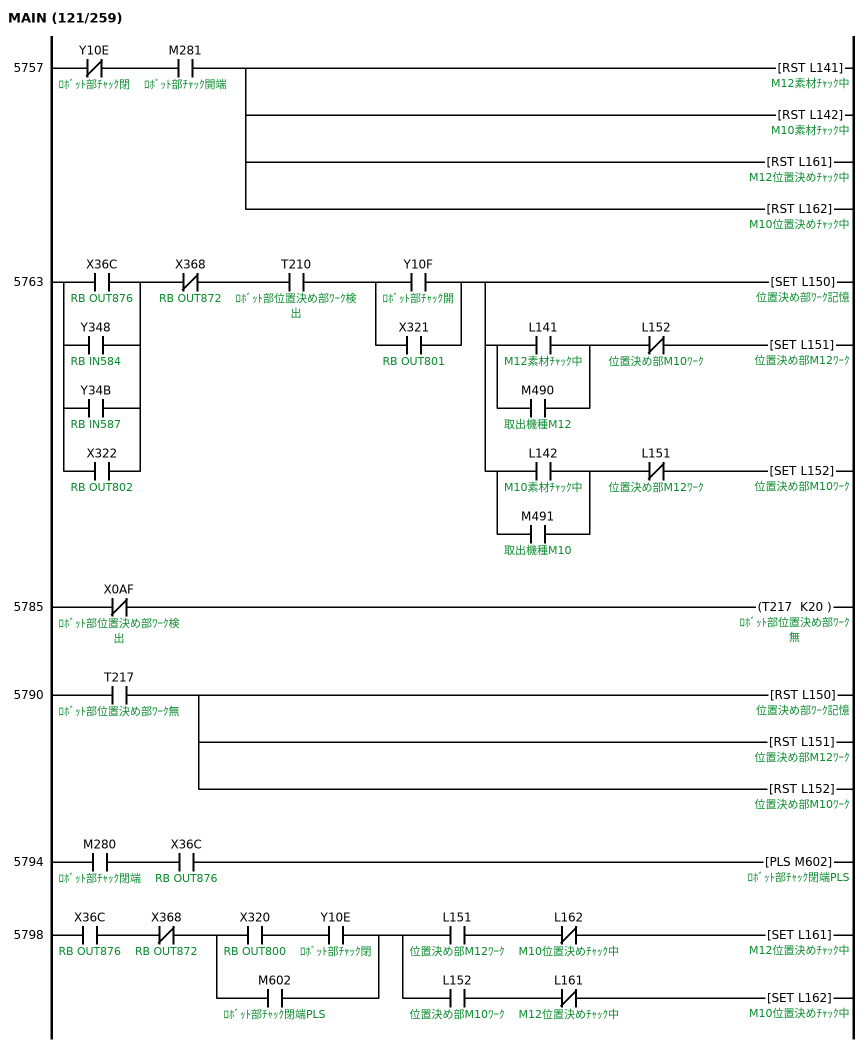
[picture p120: ladder of MAIN, rungs at steps 5757 to 5798]
5757  LDI     Y10E  ; ﾛﾎﾞｯﾄ部ﾁｬｯｸ閉
      AND     M281  ; ﾛﾎﾞｯﾄ部ﾁｬｯｸ開端
      RST     L141  ; M12素材ﾁｬｯｸ中
      RST     L142  ; M10素材ﾁｬｯｸ中
      RST     L161  ; M12位置決めﾁｬｯｸ中
      RST     L162  ; M10位置決めﾁｬｯｸ中
5763  LD      X36C  ; RB OUT876
      OR      Y348  ; RB IN584
      OR      Y34B  ; RB IN587
      OR      X322  ; RB OUT802
      ANI     X368  ; RB OUT872
      AND     T210  ; ﾛﾎﾞｯﾄ部位置決め部ﾜｰｸ検出
      LD      Y10F  ; ﾛﾎﾞｯﾄ部ﾁｬｯｸ開
      OR      X321  ; RB OUT801
      ANB
      SET     L150  ; 位置決め部ﾜｰｸ記憶
      MPS
      LD      L141  ; M12素材ﾁｬｯｸ中
      OR      M490  ; 取出機種M12
      ANB
      ANI     L152  ; 位置決め部M10ﾜｰｸ
      SET     L151  ; 位置決め部M12ﾜｰｸ
      MPP
      LD      L142  ; M10素材ﾁｬｯｸ中
      OR      M491  ; 取出機種M10
      ANB
      ANI     L151  ; 位置決め部M12ﾜｰｸ
      SET     L152  ; 位置決め部M10ﾜｰｸ
5785  LDI     X0AF  ; ﾛﾎﾞｯﾄ部位置決め部ﾜｰｸ検出
      OUT     T217 K20  ; ﾛﾎﾞｯﾄ部位置決め部ﾜｰｸ無
5790  LD      T217  ; ﾛﾎﾞｯﾄ部位置決め部ﾜｰｸ無
      RST     L150  ; 位置決め部ﾜｰｸ記憶
      RST     L151  ; 位置決め部M12ﾜｰｸ
      RST     L152  ; 位置決め部M10ﾜｰｸ
5794  LD      M280  ; ﾛﾎﾞｯﾄ部ﾁｬｯｸ閉端
      AND     X36C  ; RB OUT876
      PLS     M602  ; ﾛﾎﾞｯﾄ部ﾁｬｯｸ閉端PLS
5798  LD      X36C  ; RB OUT876
      ANI     X368  ; RB OUT872
      LD      X320  ; RB OUT800
      AND     Y10E  ; ﾛﾎﾞｯﾄ部ﾁｬｯｸ閉
      OR      M602  ; ﾛﾎﾞｯﾄ部ﾁｬｯｸ閉端PLS
      ANB
      MPS
      AND     L151  ; 位置決め部M12ﾜｰｸ
      ANI     L162  ; M10位置決めﾁｬｯｸ中
      SET     L161  ; M12位置決めﾁｬｯｸ中
      MPP
      AND     L152  ; 位置決め部M10ﾜｰｸ
      ANI     L161  ; M12位置決めﾁｬｯｸ中
      SET     L162  ; M10位置決めﾁｬｯｸ中
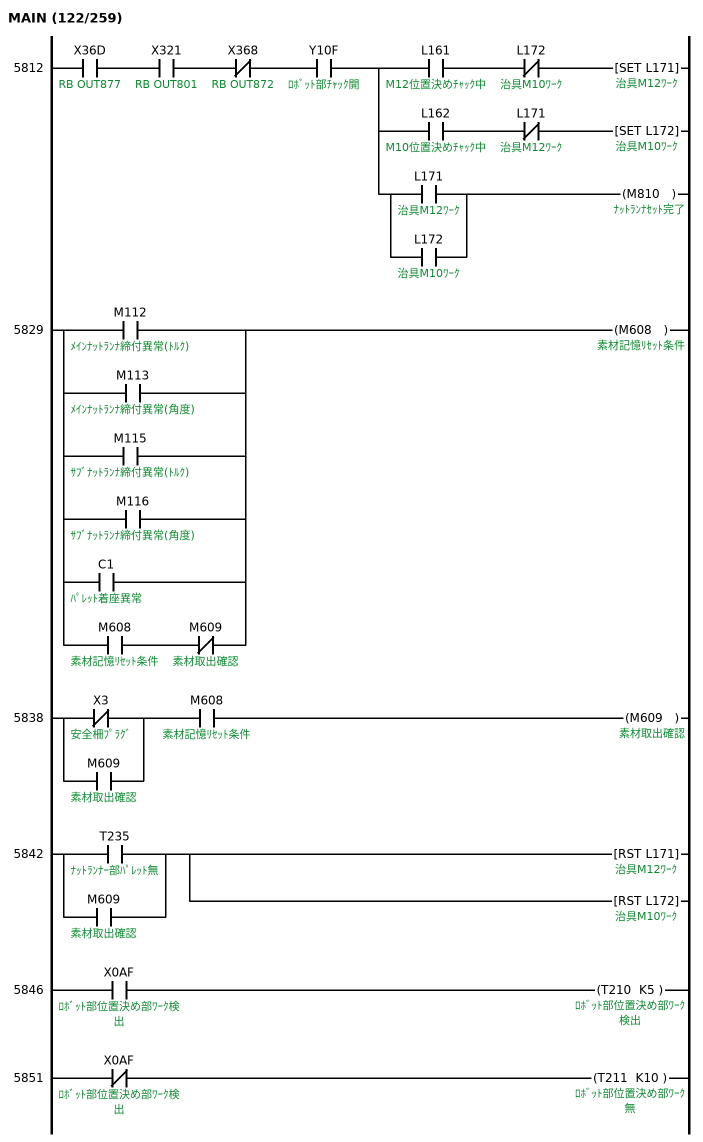
5812  LD      X36D  ; RB OUT877
      AND     X321  ; RB OUT801
      ANI     X368  ; RB OUT872
      AND     Y10F  ; ﾛﾎﾞｯﾄ部ﾁｬｯｸ開
      MPS
      AND     L161  ; M12位置決めﾁｬｯｸ中
      ANI     L172  ; 治具M10ﾜｰｸ
      SET     L171  ; 治具M12ﾜｰｸ
      MRD
      AND     L162  ; M10位置決めﾁｬｯｸ中
      ANI     L171  ; 治具M12ﾜｰｸ
      SET     L172  ; 治具M10ﾜｰｸ
      MPP
      LD      L171  ; 治具M12ﾜｰｸ
      OR      L172  ; 治具M10ﾜｰｸ
      ANB
      OUT     M810  ; ﾅｯﾄﾗﾝﾅｾｯﾄ完了
5829  LD      M112  ; ﾒｲﾝﾅｯﾄﾗﾝﾅ締付異常(ﾄﾙｸ)
      OR      M113  ; ﾒｲﾝﾅｯﾄﾗﾝﾅ締付異常(角度)
      OR      M115  ; ｻﾌﾞﾅｯﾄﾗﾝﾅ締付異常(ﾄﾙｸ)
      OR      M116  ; ｻﾌﾞﾅｯﾄﾗﾝﾅ締付異常(角度)
      OR      C1  ; ﾊﾟﾚｯﾄ着座異常
      LD      M608  ; 素材記憶ﾘｾｯﾄ条件
      ANI     M609  ; 素材取出確認
      ORB
      OUT     M608  ; 素材記憶ﾘｾｯﾄ条件
5838  LDI     X3  ; 安全柵ﾌﾟﾗｸﾞ
      OR      M609  ; 素材取出確認
      AND     M608  ; 素材記憶ﾘｾｯﾄ条件
      OUT     M609  ; 素材取出確認
5842  LD      T235  ; ﾅｯﾄﾗﾝﾅｰ部ﾊﾟﾚｯﾄ無
      OR      M609  ; 素材取出確認
      RST     L171  ; 治具M12ﾜｰｸ
      RST     L172  ; 治具M10ﾜｰｸ
5846  LD      X0AF  ; ﾛﾎﾞｯﾄ部位置決め部ﾜｰｸ検出
      OUT     T210 K5  ; ﾛﾎﾞｯﾄ部位置決め部ﾜｰｸ検出
5851  LDI     X0AF  ; ﾛﾎﾞｯﾄ部位置決め部ﾜｰｸ検出
      OUT     T211 K10  ; ﾛﾎﾞｯﾄ部位置決め部ﾜｰｸ無
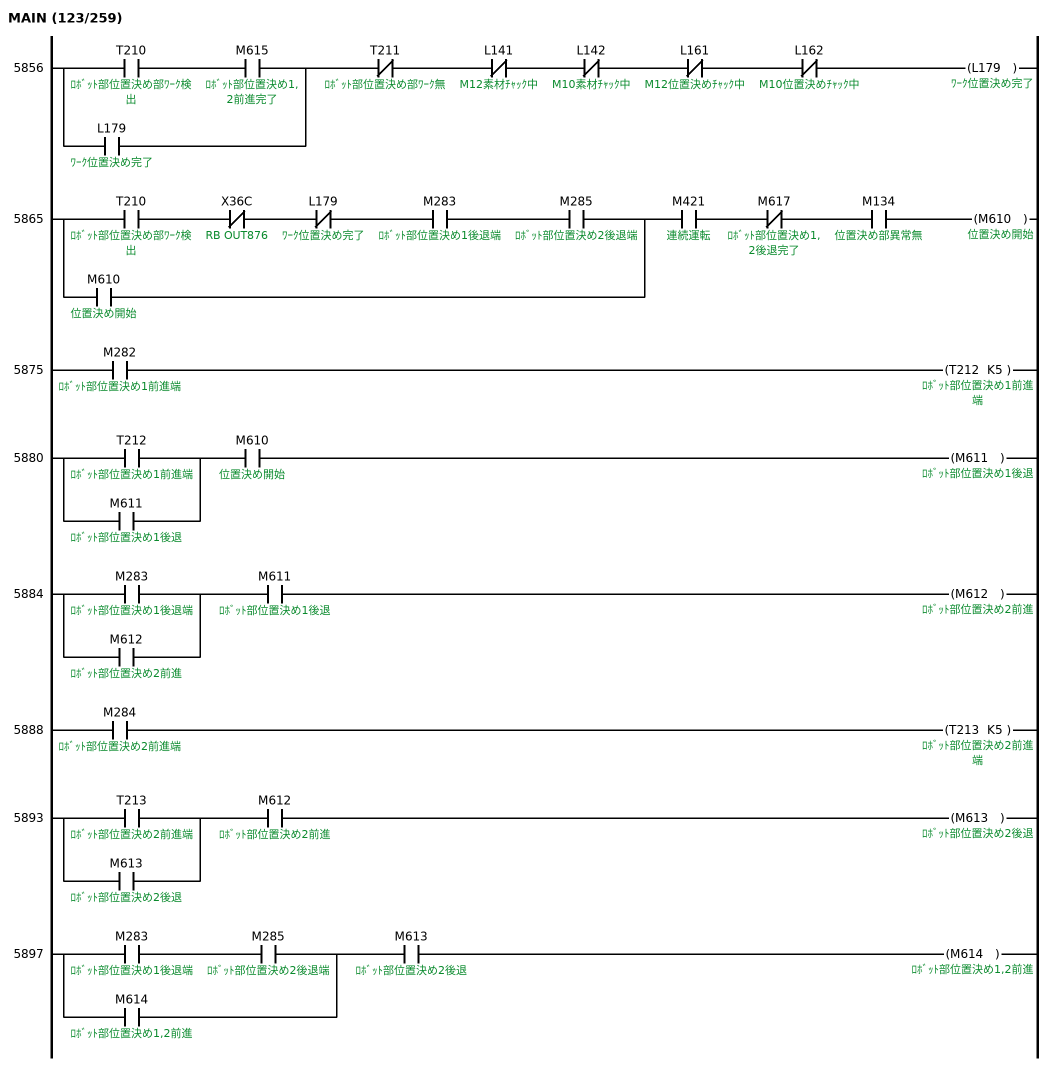
5856  LD      T210  ; ﾛﾎﾞｯﾄ部位置決め部ﾜｰｸ検出
      AND     M615  ; ﾛﾎﾞｯﾄ部位置決め1,2前進完了
      OR      L179  ; ﾜｰｸ位置決め完了
      ANI     T211  ; ﾛﾎﾞｯﾄ部位置決め部ﾜｰｸ無
      ANI     L141  ; M12素材ﾁｬｯｸ中
      ANI     L142  ; M10素材ﾁｬｯｸ中
      ANI     L161  ; M12位置決めﾁｬｯｸ中
      ANI     L162  ; M10位置決めﾁｬｯｸ中
      OUT     L179  ; ﾜｰｸ位置決め完了
5865  LD      T210  ; ﾛﾎﾞｯﾄ部位置決め部ﾜｰｸ検出
      ANI     X36C  ; RB OUT876
      ANI     L179  ; ﾜｰｸ位置決め完了
      AND     M283  ; ﾛﾎﾞｯﾄ部位置決め1後退端
      AND     M285  ; ﾛﾎﾞｯﾄ部位置決め2後退端
      OR      M610  ; 位置決め開始
      AND     M421  ; 連続運転
      ANI     M617  ; ﾛﾎﾞｯﾄ部位置決め1,2後退完了
      AND     M134  ; 位置決め部異常無
      OUT     M610  ; 位置決め開始
5875  LD      M282  ; ﾛﾎﾞｯﾄ部位置決め1前進端
      OUT     T212 K5  ; ﾛﾎﾞｯﾄ部位置決め1前進端
5880  LD      T212  ; ﾛﾎﾞｯﾄ部位置決め1前進端
      OR      M611  ; ﾛﾎﾞｯﾄ部位置決め1後退
      AND     M610  ; 位置決め開始
      OUT     M611  ; ﾛﾎﾞｯﾄ部位置決め1後退
5884  LD      M283  ; ﾛﾎﾞｯﾄ部位置決め1後退端
      OR      M612  ; ﾛﾎﾞｯﾄ部位置決め2前進
      AND     M611  ; ﾛﾎﾞｯﾄ部位置決め1後退
      OUT     M612  ; ﾛﾎﾞｯﾄ部位置決め2前進
5888  LD      M284  ; ﾛﾎﾞｯﾄ部位置決め2前進端
      OUT     T213 K5  ; ﾛﾎﾞｯﾄ部位置決め2前進端
5893  LD      T213  ; ﾛﾎﾞｯﾄ部位置決め2前進端
      OR      M613  ; ﾛﾎﾞｯﾄ部位置決め2後退
      AND     M612  ; ﾛﾎﾞｯﾄ部位置決め2前進
      OUT     M613  ; ﾛﾎﾞｯﾄ部位置決め2後退
5897  LD      M283  ; ﾛﾎﾞｯﾄ部位置決め1後退端
      AND     M285  ; ﾛﾎﾞｯﾄ部位置決め2後退端
      OR      M614  ; ﾛﾎﾞｯﾄ部位置決め1,2前進
      AND     M613  ; ﾛﾎﾞｯﾄ部位置決め2後退
      OUT     M614  ; ﾛﾎﾞｯﾄ部位置決め1,2前進
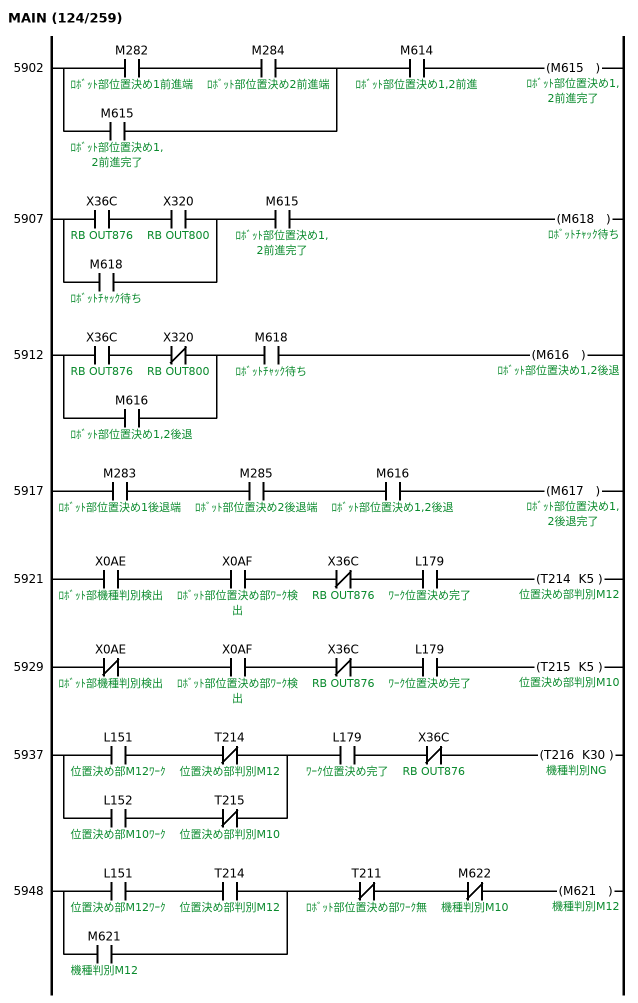
5902  LD      M282  ; ﾛﾎﾞｯﾄ部位置決め1前進端
      AND     M284  ; ﾛﾎﾞｯﾄ部位置決め2前進端
      OR      M615  ; ﾛﾎﾞｯﾄ部位置決め1,2前進完了
      AND     M614  ; ﾛﾎﾞｯﾄ部位置決め1,2前進
      OUT     M615  ; ﾛﾎﾞｯﾄ部位置決め1,2前進完了
5907  LD      X36C  ; RB OUT876
      AND     X320  ; RB OUT800
      OR      M618  ; ﾛﾎﾞｯﾄﾁｬｯｸ待ち
      AND     M615  ; ﾛﾎﾞｯﾄ部位置決め1,2前進完了
      OUT     M618  ; ﾛﾎﾞｯﾄﾁｬｯｸ待ち
5912  LD      X36C  ; RB OUT876
      ANI     X320  ; RB OUT800
      OR      M616  ; ﾛﾎﾞｯﾄ部位置決め1,2後退
      AND     M618  ; ﾛﾎﾞｯﾄﾁｬｯｸ待ち
      OUT     M616  ; ﾛﾎﾞｯﾄ部位置決め1,2後退
5917  LD      M283  ; ﾛﾎﾞｯﾄ部位置決め1後退端
      AND     M285  ; ﾛﾎﾞｯﾄ部位置決め2後退端
      AND     M616  ; ﾛﾎﾞｯﾄ部位置決め1,2後退
      OUT     M617  ; ﾛﾎﾞｯﾄ部位置決め1,2後退完了
5921  LD      X0AE  ; ﾛﾎﾞｯﾄ部機種判別検出
      AND     X0AF  ; ﾛﾎﾞｯﾄ部位置決め部ﾜｰｸ検出
      ANI     X36C  ; RB OUT876
      AND     L179  ; ﾜｰｸ位置決め完了
      OUT     T214 K5  ; 位置決め部判別M12
5929  LDI     X0AE  ; ﾛﾎﾞｯﾄ部機種判別検出
      AND     X0AF  ; ﾛﾎﾞｯﾄ部位置決め部ﾜｰｸ検出
      ANI     X36C  ; RB OUT876
      AND     L179  ; ﾜｰｸ位置決め完了
      OUT     T215 K5  ; 位置決め部判別M10
5937  LD      L151  ; 位置決め部M12ﾜｰｸ
      ANI     T214  ; 位置決め部判別M12
      LD      L152  ; 位置決め部M10ﾜｰｸ
      ANI     T215  ; 位置決め部判別M10
      ORB
      AND     L179  ; ﾜｰｸ位置決め完了
      ANI     X36C  ; RB OUT876
      OUT     T216 K30  ; 機種判別NG
5948  LD      L151  ; 位置決め部M12ﾜｰｸ
      AND     T214  ; 位置決め部判別M12
      OR      M621  ; 機種判別M12
      ANI     T211  ; ﾛﾎﾞｯﾄ部位置決め部ﾜｰｸ無
      ANI     M622  ; 機種判別M10
      OUT     M621  ; 機種判別M12
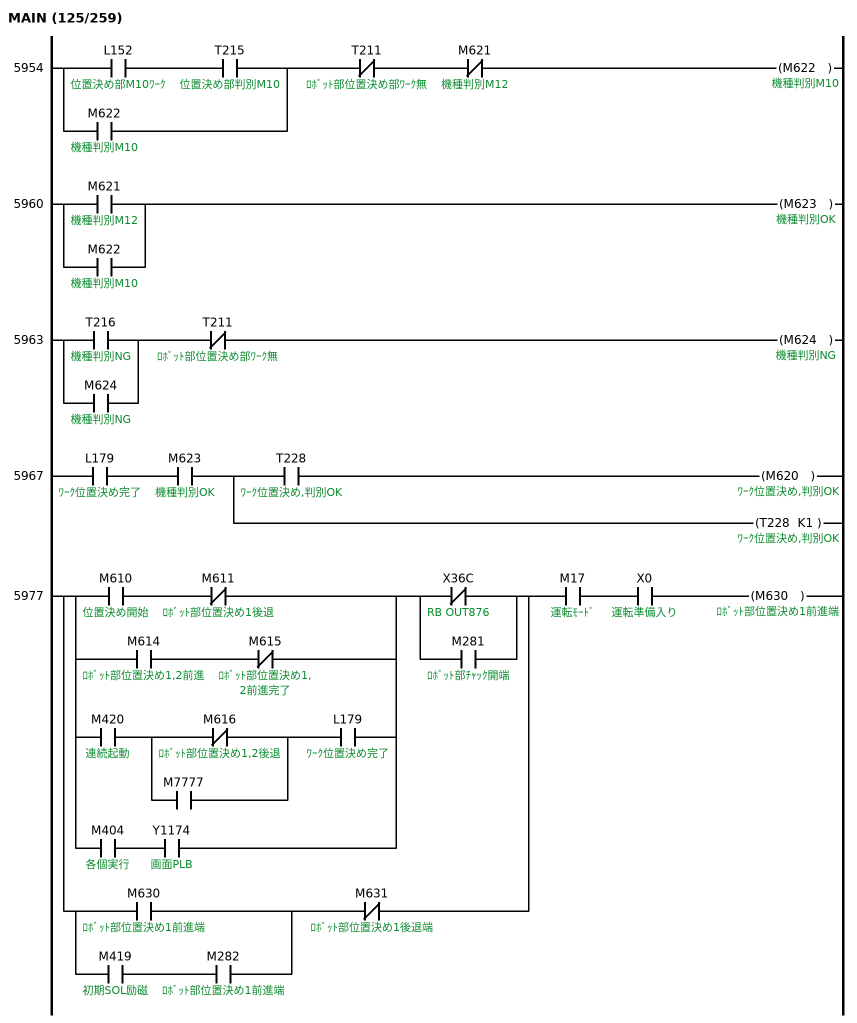
5954  LD      L152  ; 位置決め部M10ﾜｰｸ
      AND     T215  ; 位置決め部判別M10
      OR      M622  ; 機種判別M10
      ANI     T211  ; ﾛﾎﾞｯﾄ部位置決め部ﾜｰｸ無
      ANI     M621  ; 機種判別M12
      OUT     M622  ; 機種判別M10
5960  LD      M621  ; 機種判別M12
      OR      M622  ; 機種判別M10
      OUT     M623  ; 機種判別OK
5963  LD      T216  ; 機種判別NG
      OR      M624  ; 機種判別NG
      ANI     T211  ; ﾛﾎﾞｯﾄ部位置決め部ﾜｰｸ無
      OUT     M624  ; 機種判別NG
5967  LD      L179  ; ﾜｰｸ位置決め完了
      AND     M623  ; 機種判別OK
      MPS
      AND     T228  ; ﾜｰｸ位置決め,判別OK
      OUT     M620  ; ﾜｰｸ位置決め,判別OK
      MPP
      OUT     T228 K1  ; ﾜｰｸ位置決め,判別OK
5977  LD      M610  ; 位置決め開始
      ANI     M611  ; ﾛﾎﾞｯﾄ部位置決め1後退
      LD      M614  ; ﾛﾎﾞｯﾄ部位置決め1,2前進
      ANI     M615  ; ﾛﾎﾞｯﾄ部位置決め1,2前進完了
      ORB
      LD      M420  ; 連続起動
      LDI     M616  ; ﾛﾎﾞｯﾄ部位置決め1,2後退
      OR      M7777
      ANB
      AND     L179  ; ﾜｰｸ位置決め完了
      ORB
      LD      M404  ; 各個実行
      AND     Y1174  ; 画面PLB
      ORB
      LDI     X36C  ; RB OUT876
      OR      M281  ; ﾛﾎﾞｯﾄ部ﾁｬｯｸ開端
      ANB
      LD      M630  ; ﾛﾎﾞｯﾄ部位置決め1前進端
      LD      M419  ; 初期SOL励磁
      AND     M282  ; ﾛﾎﾞｯﾄ部位置決め1前進端
      ORB
      ANI     M631  ; ﾛﾎﾞｯﾄ部位置決め1後退端
      ORB
      AND     M17  ; 運転ﾓｰﾄﾞ
      AND     X0  ; 運転準備入り
      OUT     M630  ; ﾛﾎﾞｯﾄ部位置決め1前進端
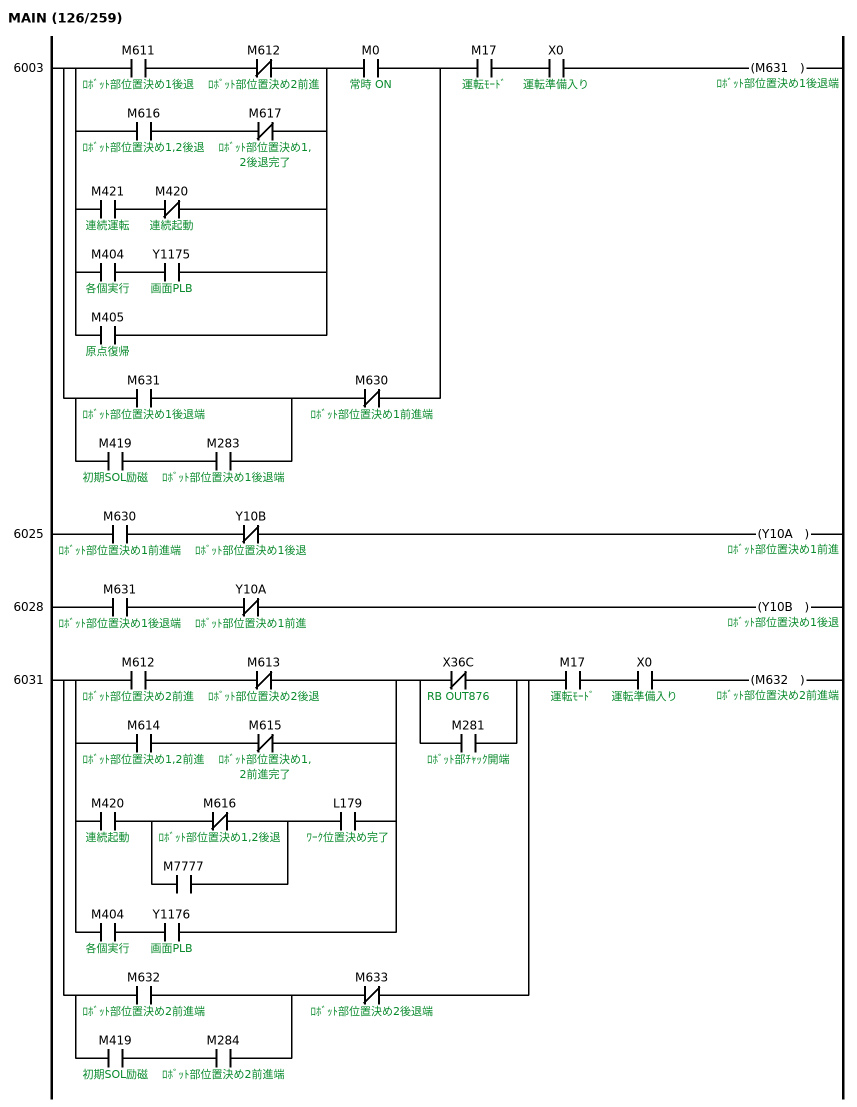
6003  LD      M611  ; ﾛﾎﾞｯﾄ部位置決め1後退
      ANI     M612  ; ﾛﾎﾞｯﾄ部位置決め2前進
      LD      M616  ; ﾛﾎﾞｯﾄ部位置決め1,2後退
      ANI     M617  ; ﾛﾎﾞｯﾄ部位置決め1,2後退完了
      ORB
      LD      M421  ; 連続運転
      ANI     M420  ; 連続起動
      ORB
      LD      M404  ; 各個実行
      AND     Y1175  ; 画面PLB
      ORB
      OR      M405  ; 原点復帰
      AND     M0  ; 常時 ON
      LD      M631  ; ﾛﾎﾞｯﾄ部位置決め1後退端
      LD      M419  ; 初期SOL励磁
      AND     M283  ; ﾛﾎﾞｯﾄ部位置決め1後退端
      ORB
      ANI     M630  ; ﾛﾎﾞｯﾄ部位置決め1前進端
      ORB
      AND     M17  ; 運転ﾓｰﾄﾞ
      AND     X0  ; 運転準備入り
      OUT     M631  ; ﾛﾎﾞｯﾄ部位置決め1後退端
6025  LD      M630  ; ﾛﾎﾞｯﾄ部位置決め1前進端
      ANI     Y10B  ; ﾛﾎﾞｯﾄ部位置決め1後退
      OUT     Y10A  ; ﾛﾎﾞｯﾄ部位置決め1前進
6028  LD      M631  ; ﾛﾎﾞｯﾄ部位置決め1後退端
      ANI     Y10A  ; ﾛﾎﾞｯﾄ部位置決め1前進
      OUT     Y10B  ; ﾛﾎﾞｯﾄ部位置決め1後退
6031  LD      M612  ; ﾛﾎﾞｯﾄ部位置決め2前進
      ANI     M613  ; ﾛﾎﾞｯﾄ部位置決め2後退
      LD      M614  ; ﾛﾎﾞｯﾄ部位置決め1,2前進
      ANI     M615  ; ﾛﾎﾞｯﾄ部位置決め1,2前進完了
      ORB
      LD      M420  ; 連続起動
      LDI     M616  ; ﾛﾎﾞｯﾄ部位置決め1,2後退
      OR      M7777
      ANB
      AND     L179  ; ﾜｰｸ位置決め完了
      ORB
      LD      M404  ; 各個実行
      AND     Y1176  ; 画面PLB
      ORB
      LDI     X36C  ; RB OUT876
      OR      M281  ; ﾛﾎﾞｯﾄ部ﾁｬｯｸ開端
      ANB
      LD      M632  ; ﾛﾎﾞｯﾄ部位置決め2前進端
      LD      M419  ; 初期SOL励磁
      AND     M284  ; ﾛﾎﾞｯﾄ部位置決め2前進端
      ORB
      ANI     M633  ; ﾛﾎﾞｯﾄ部位置決め2後退端
      ORB
      AND     M17  ; 運転ﾓｰﾄﾞ
      AND     X0  ; 運転準備入り
      OUT     M632  ; ﾛﾎﾞｯﾄ部位置決め2前進端
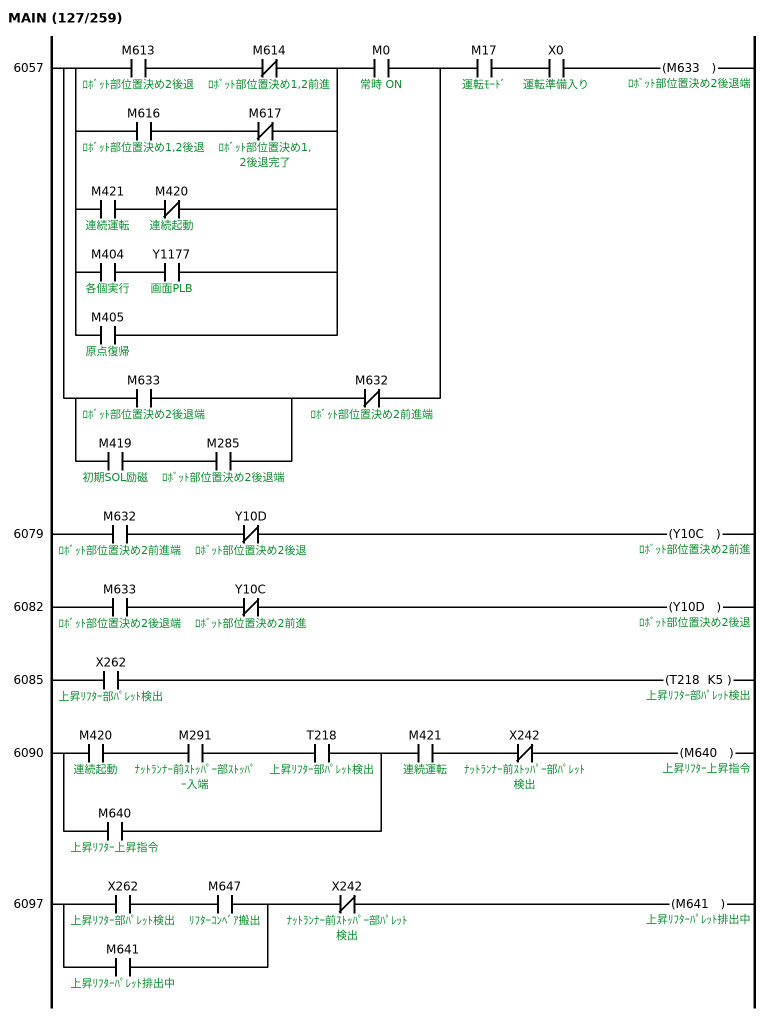
6057  LD      M613  ; ﾛﾎﾞｯﾄ部位置決め2後退
      ANI     M614  ; ﾛﾎﾞｯﾄ部位置決め1,2前進
      LD      M616  ; ﾛﾎﾞｯﾄ部位置決め1,2後退
      ANI     M617  ; ﾛﾎﾞｯﾄ部位置決め1,2後退完了
      ORB
      LD      M421  ; 連続運転
      ANI     M420  ; 連続起動
      ORB
      LD      M404  ; 各個実行
      AND     Y1177  ; 画面PLB
      ORB
      OR      M405  ; 原点復帰
      AND     M0  ; 常時 ON
      LD      M633  ; ﾛﾎﾞｯﾄ部位置決め2後退端
      LD      M419  ; 初期SOL励磁
      AND     M285  ; ﾛﾎﾞｯﾄ部位置決め2後退端
      ORB
      ANI     M632  ; ﾛﾎﾞｯﾄ部位置決め2前進端
      ORB
      AND     M17  ; 運転ﾓｰﾄﾞ
      AND     X0  ; 運転準備入り
      OUT     M633  ; ﾛﾎﾞｯﾄ部位置決め2後退端
6079  LD      M632  ; ﾛﾎﾞｯﾄ部位置決め2前進端
      ANI     Y10D  ; ﾛﾎﾞｯﾄ部位置決め2後退
      OUT     Y10C  ; ﾛﾎﾞｯﾄ部位置決め2前進
6082  LD      M633  ; ﾛﾎﾞｯﾄ部位置決め2後退端
      ANI     Y10C  ; ﾛﾎﾞｯﾄ部位置決め2前進
      OUT     Y10D  ; ﾛﾎﾞｯﾄ部位置決め2後退
6085  LD      X262  ; 上昇ﾘﾌﾀｰ部ﾊﾟﾚｯﾄ検出
      OUT     T218 K5  ; 上昇ﾘﾌﾀｰ部ﾊﾟﾚｯﾄ検出
6090  LD      M420  ; 連続起動
      AND     M291  ; ﾅｯﾄﾗﾝﾅｰ前ｽﾄｯﾊﾟｰ部ｽﾄｯﾊﾟｰ入端
      AND     T218  ; 上昇ﾘﾌﾀｰ部ﾊﾟﾚｯﾄ検出
      OR      M640  ; 上昇ﾘﾌﾀｰ上昇指令
      AND     M421  ; 連続運転
      ANI     X242  ; ﾅｯﾄﾗﾝﾅｰ前ｽﾄｯﾊﾟｰ部ﾊﾟﾚｯﾄ検出
      OUT     M640  ; 上昇ﾘﾌﾀｰ上昇指令
6097  LD      X262  ; 上昇ﾘﾌﾀｰ部ﾊﾟﾚｯﾄ検出
      AND     M647  ; ﾘﾌﾀｰｺﾝﾍﾞｱ搬出
      OR      M641  ; 上昇ﾘﾌﾀｰﾊﾟﾚｯﾄ排出中
      ANI     X242  ; ﾅｯﾄﾗﾝﾅｰ前ｽﾄｯﾊﾟｰ部ﾊﾟﾚｯﾄ検出
      OUT     M641  ; 上昇ﾘﾌﾀｰﾊﾟﾚｯﾄ排出中
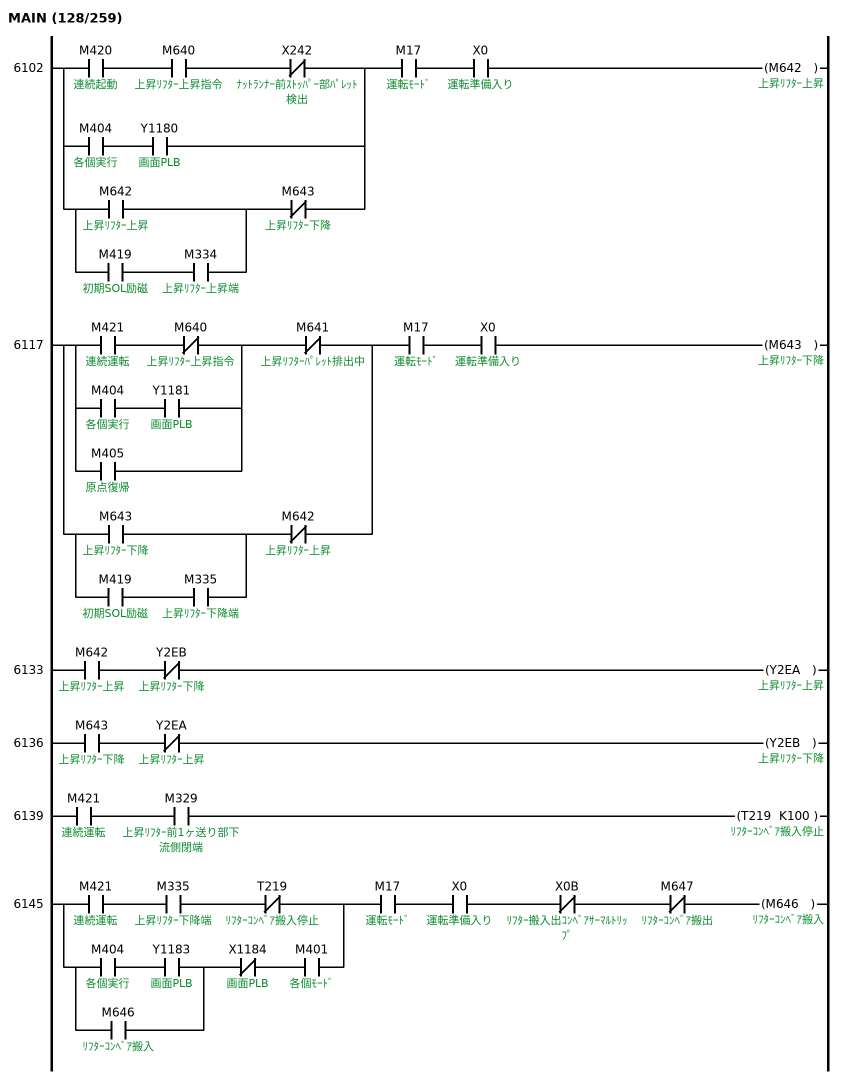
6102  LD      M420  ; 連続起動
      AND     M640  ; 上昇ﾘﾌﾀｰ上昇指令
      ANI     X242  ; ﾅｯﾄﾗﾝﾅｰ前ｽﾄｯﾊﾟｰ部ﾊﾟﾚｯﾄ検出
      LD      M404  ; 各個実行
      AND     Y1180  ; 画面PLB
      ORB
      LD      M642  ; 上昇ﾘﾌﾀｰ上昇
      LD      M419  ; 初期SOL励磁
      AND     M334  ; 上昇ﾘﾌﾀｰ上昇端
      ORB
      ANI     M643  ; 上昇ﾘﾌﾀｰ下降
      ORB
      AND     M17  ; 運転ﾓｰﾄﾞ
      AND     X0  ; 運転準備入り
      OUT     M642  ; 上昇ﾘﾌﾀｰ上昇
6117  LD      M421  ; 連続運転
      ANI     M640  ; 上昇ﾘﾌﾀｰ上昇指令
      LD      M404  ; 各個実行
      AND     Y1181  ; 画面PLB
      ORB
      OR      M405  ; 原点復帰
      ANI     M641  ; 上昇ﾘﾌﾀｰﾊﾟﾚｯﾄ排出中
      LD      M643  ; 上昇ﾘﾌﾀｰ下降
      LD      M419  ; 初期SOL励磁
      AND     M335  ; 上昇ﾘﾌﾀｰ下降端
      ORB
      ANI     M642  ; 上昇ﾘﾌﾀｰ上昇
      ORB
      AND     M17  ; 運転ﾓｰﾄﾞ
      AND     X0  ; 運転準備入り
      OUT     M643  ; 上昇ﾘﾌﾀｰ下降
6133  LD      M642  ; 上昇ﾘﾌﾀｰ上昇
      ANI     Y2EB  ; 上昇ﾘﾌﾀｰ下降
      OUT     Y2EA  ; 上昇ﾘﾌﾀｰ上昇
6136  LD      M643  ; 上昇ﾘﾌﾀｰ下降
      ANI     Y2EA  ; 上昇ﾘﾌﾀｰ上昇
      OUT     Y2EB  ; 上昇ﾘﾌﾀｰ下降
6139  LD      M421  ; 連続運転
      AND     M329  ; 上昇ﾘﾌﾀｰ前1ヶ送り部下流側閉端
      OUT     T219 K100  ; ﾘﾌﾀｰｺﾝﾍﾞｱ搬入停止
6145  LD      M421  ; 連続運転
      AND     M335  ; 上昇ﾘﾌﾀｰ下降端
      ANI     T219  ; ﾘﾌﾀｰｺﾝﾍﾞｱ搬入停止
      LD      M404  ; 各個実行
      AND     Y1183  ; 画面PLB
      OR      M646  ; ﾘﾌﾀｰｺﾝﾍﾞｱ搬入
      ANI     X1184  ; 画面PLB
      AND     M401  ; 各個ﾓｰﾄﾞ
      ORB
      AND     M17  ; 運転ﾓｰﾄﾞ
      AND     X0  ; 運転準備入り
      ANI     X0B  ; ﾘﾌﾀｰ搬入出ｺﾝﾍﾞｱｻｰﾏﾙﾄﾘｯﾌﾟ
      ANI     M647  ; ﾘﾌﾀｰｺﾝﾍﾞｱ搬出
      OUT     M646  ; ﾘﾌﾀｰｺﾝﾍﾞｱ搬入
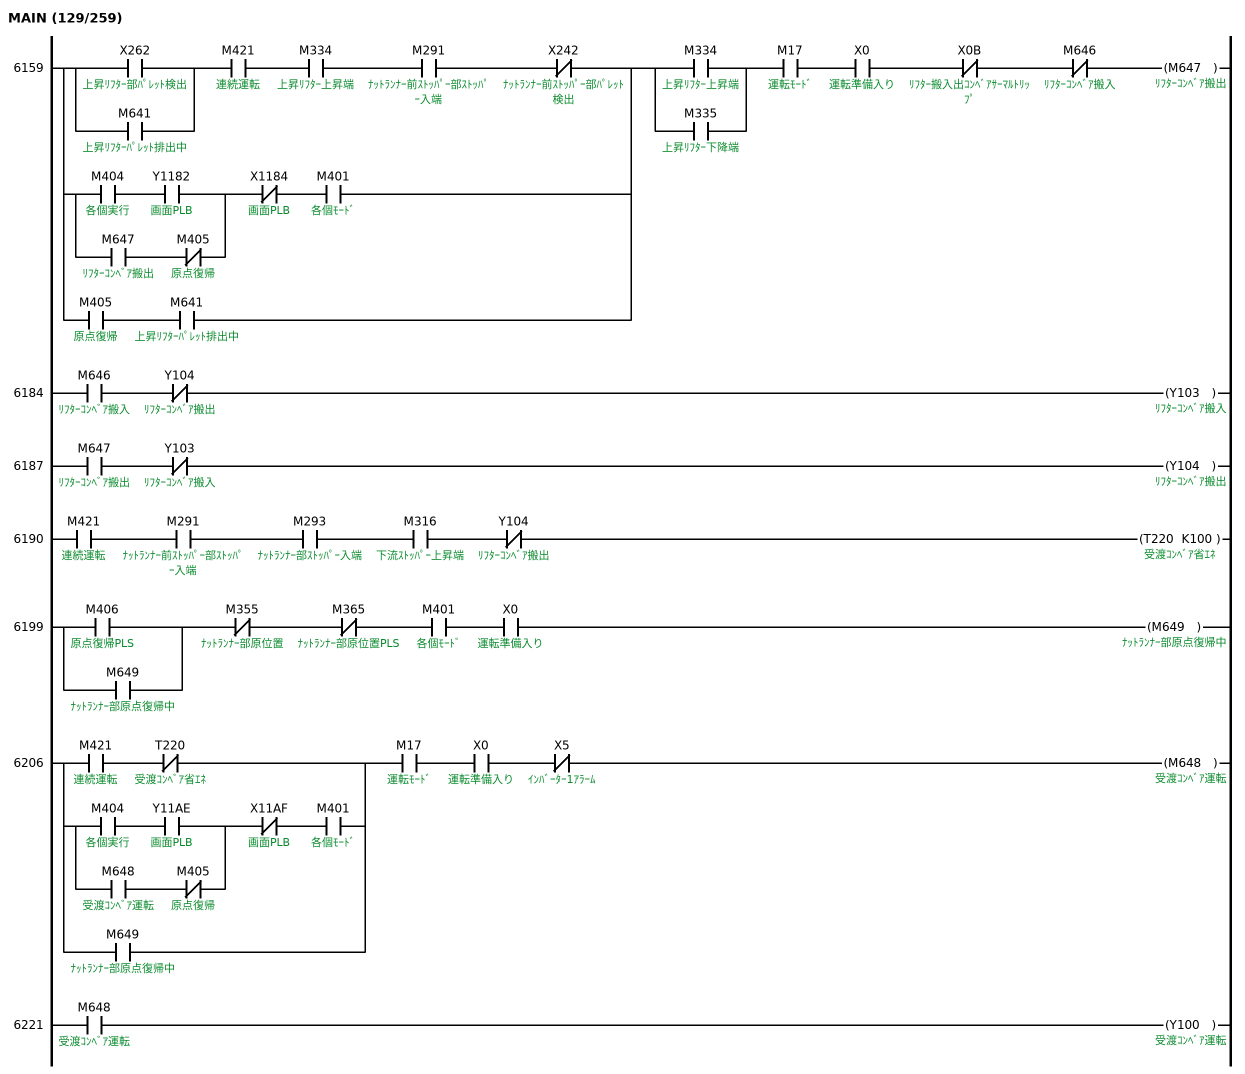
6159  LD      X262  ; 上昇ﾘﾌﾀｰ部ﾊﾟﾚｯﾄ検出
      OR      M641  ; 上昇ﾘﾌﾀｰﾊﾟﾚｯﾄ排出中
      AND     M421  ; 連続運転
      AND     M334  ; 上昇ﾘﾌﾀｰ上昇端
      AND     M291  ; ﾅｯﾄﾗﾝﾅｰ前ｽﾄｯﾊﾟｰ部ｽﾄｯﾊﾟｰ入端
      ANI     X242  ; ﾅｯﾄﾗﾝﾅｰ前ｽﾄｯﾊﾟｰ部ﾊﾟﾚｯﾄ検出
      LD      M404  ; 各個実行
      AND     Y1182  ; 画面PLB
      LD      M647  ; ﾘﾌﾀｰｺﾝﾍﾞｱ搬出
      ANI     M405  ; 原点復帰
      ORB
      ANI     X1184  ; 画面PLB
      AND     M401  ; 各個ﾓｰﾄﾞ
      ORB
      LD      M405  ; 原点復帰
      AND     M641  ; 上昇ﾘﾌﾀｰﾊﾟﾚｯﾄ排出中
      ORB
      LD      M334  ; 上昇ﾘﾌﾀｰ上昇端
      OR      M335  ; 上昇ﾘﾌﾀｰ下降端
      ANB
      AND     M17  ; 運転ﾓｰﾄﾞ
      AND     X0  ; 運転準備入り
      ANI     X0B  ; ﾘﾌﾀｰ搬入出ｺﾝﾍﾞｱｻｰﾏﾙﾄﾘｯﾌﾟ
      ANI     M646  ; ﾘﾌﾀｰｺﾝﾍﾞｱ搬入
      OUT     M647  ; ﾘﾌﾀｰｺﾝﾍﾞｱ搬出
6184  LD      M646  ; ﾘﾌﾀｰｺﾝﾍﾞｱ搬入
      ANI     Y104  ; ﾘﾌﾀｰｺﾝﾍﾞｱ搬出
      OUT     Y103  ; ﾘﾌﾀｰｺﾝﾍﾞｱ搬入
6187  LD      M647  ; ﾘﾌﾀｰｺﾝﾍﾞｱ搬出
      ANI     Y103  ; ﾘﾌﾀｰｺﾝﾍﾞｱ搬入
      OUT     Y104  ; ﾘﾌﾀｰｺﾝﾍﾞｱ搬出
6190  LD      M421  ; 連続運転
      AND     M291  ; ﾅｯﾄﾗﾝﾅｰ前ｽﾄｯﾊﾟｰ部ｽﾄｯﾊﾟｰ入端
      AND     M293  ; ﾅｯﾄﾗﾝﾅｰ部ｽﾄｯﾊﾟｰ入端
      AND     M316  ; 下流ｽﾄｯﾊﾟｰ上昇端
      ANI     Y104  ; ﾘﾌﾀｰｺﾝﾍﾞｱ搬出
      OUT     T220 K100  ; 受渡ｺﾝﾍﾞｱ省ｴﾈ
6199  LD      M406  ; 原点復帰PLS
      OR      M649  ; ﾅｯﾄﾗﾝﾅｰ部原点復帰中
      ANI     M355  ; ﾅｯﾄﾗﾝﾅｰ部原位置
      ANI     M365  ; ﾅｯﾄﾗﾝﾅｰ部原位置PLS
      AND     M401  ; 各個ﾓｰﾄﾞ
      AND     X0  ; 運転準備入り
      OUT     M649  ; ﾅｯﾄﾗﾝﾅｰ部原点復帰中
6206  LD      M421  ; 連続運転
      ANI     T220  ; 受渡ｺﾝﾍﾞｱ省ｴﾈ
      LD      M404  ; 各個実行
      AND     Y11AE  ; 画面PLB
      LD      M648  ; 受渡ｺﾝﾍﾞｱ運転
      ANI     M405  ; 原点復帰
      ORB
      ANI     X11AF  ; 画面PLB
      AND     M401  ; 各個ﾓｰﾄﾞ
      ORB
      OR      M649  ; ﾅｯﾄﾗﾝﾅｰ部原点復帰中
      AND     M17  ; 運転ﾓｰﾄﾞ
      AND     X0  ; 運転準備入り
      ANI     X5  ; ｲﾝﾊﾞｰﾀｰ1ｱﾗｰﾑ
      OUT     M648  ; 受渡ｺﾝﾍﾞｱ運転
6221  LD      M648  ; 受渡ｺﾝﾍﾞｱ運転
      OUT     Y100  ; 受渡ｺﾝﾍﾞｱ運転
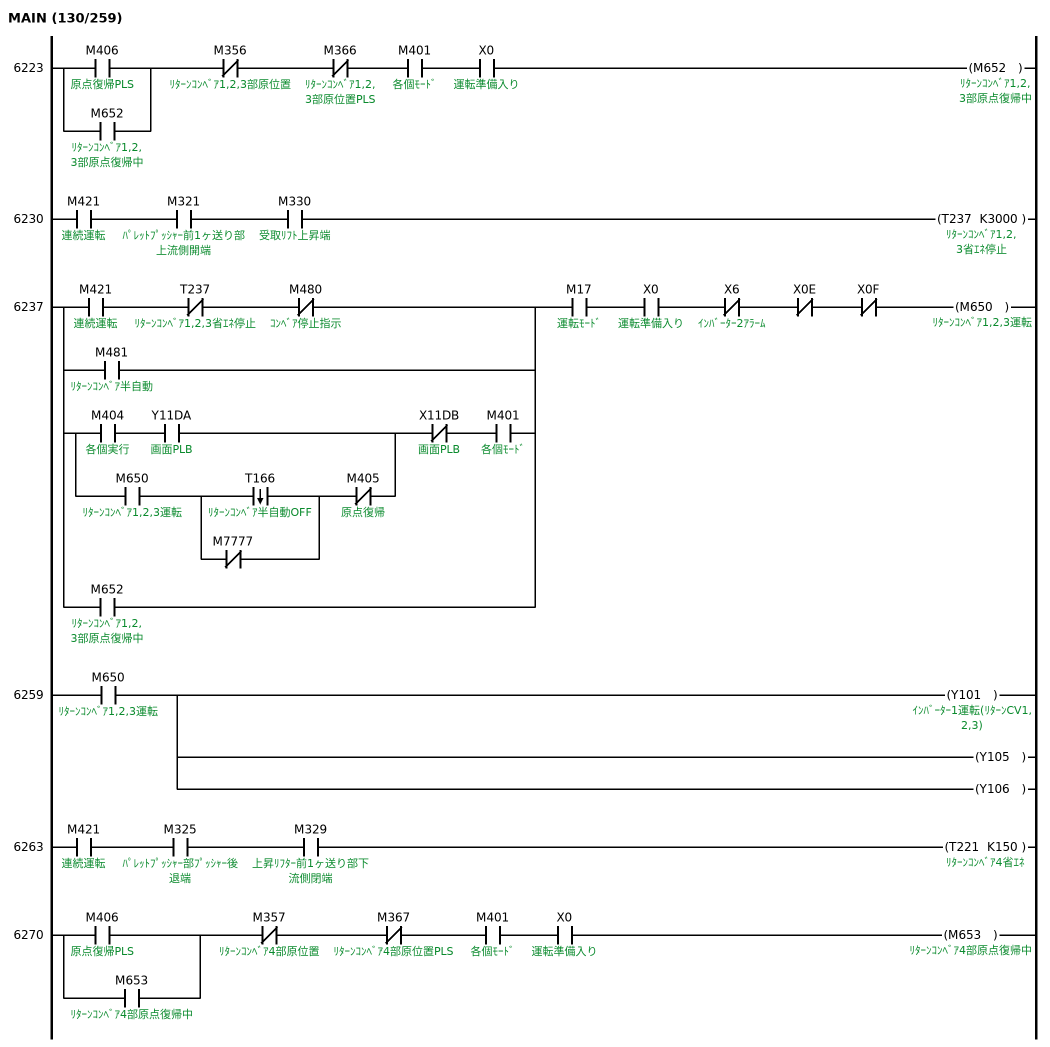
6223  LD      M406  ; 原点復帰PLS
      OR      M652  ; ﾘﾀｰﾝｺﾝﾍﾞｱ1,2,3部原点復帰中
      ANI     M356  ; ﾘﾀｰﾝｺﾝﾍﾞｱ1,2,3部原位置
      ANI     M366  ; ﾘﾀｰﾝｺﾝﾍﾞｱ1,2,3部原位置PLS
      AND     M401  ; 各個ﾓｰﾄﾞ
      AND     X0  ; 運転準備入り
      OUT     M652  ; ﾘﾀｰﾝｺﾝﾍﾞｱ1,2,3部原点復帰中
6230  LD      M421  ; 連続運転
      AND     M321  ; ﾊﾟﾚｯﾄﾌﾟｯｼｬｰ前1ヶ送り部上流側開端
      AND     M330  ; 受取ﾘﾌﾄ上昇端
      OUT     T237 K3000  ; ﾘﾀｰﾝｺﾝﾍﾞｱ1,2,3省ｴﾈ停止
6237  LD      M421  ; 連続運転
      ANI     T237  ; ﾘﾀｰﾝｺﾝﾍﾞｱ1,2,3省ｴﾈ停止
      ANI     M480  ; ｺﾝﾍﾞｱ停止指示
      OR      M481  ; ﾘﾀｰﾝｺﾝﾍﾞｱ半自動
      LD      M404  ; 各個実行
      AND     Y11DA  ; 画面PLB
      LD      M650  ; ﾘﾀｰﾝｺﾝﾍﾞｱ1,2,3運転
      LDF     T166  ; ﾘﾀｰﾝｺﾝﾍﾞｱ半自動OFF
      ORI     M7777
      ANB
      ANI     M405  ; 原点復帰
      ORB
      ANI     X11DB  ; 画面PLB
      AND     M401  ; 各個ﾓｰﾄﾞ
      ORB
      OR      M652  ; ﾘﾀｰﾝｺﾝﾍﾞｱ1,2,3部原点復帰中
      AND     M17  ; 運転ﾓｰﾄﾞ
      AND     X0  ; 運転準備入り
      ANI     X6  ; ｲﾝﾊﾞｰﾀｰ2ｱﾗｰﾑ
      ANI     X0E
      ANI     X0F
      OUT     M650  ; ﾘﾀｰﾝｺﾝﾍﾞｱ1,2,3運転
6259  LD      M650  ; ﾘﾀｰﾝｺﾝﾍﾞｱ1,2,3運転
      OUT     Y101  ; ｲﾝﾊﾞｰﾀｰ1運転(ﾘﾀｰﾝCV1,2,3)
      OUT     Y105
      OUT     Y106
6263  LD      M421  ; 連続運転
      AND     M325  ; ﾊﾟﾚｯﾄﾌﾟｯｼｬｰ部ﾌﾟｯｼｬｰ後退端
      AND     M329  ; 上昇ﾘﾌﾀｰ前1ヶ送り部下流側閉端
      OUT     T221 K150  ; ﾘﾀｰﾝｺﾝﾍﾞｱ4省ｴﾈ
6270  LD      M406  ; 原点復帰PLS
      OR      M653  ; ﾘﾀｰﾝｺﾝﾍﾞｱ4部原点復帰中
      ANI     M357  ; ﾘﾀｰﾝｺﾝﾍﾞｱ4部原位置
      ANI     M367  ; ﾘﾀｰﾝｺﾝﾍﾞｱ4部原位置PLS
      AND     M401  ; 各個ﾓｰﾄﾞ
      AND     X0  ; 運転準備入り
      OUT     M653  ; ﾘﾀｰﾝｺﾝﾍﾞｱ4部原点復帰中
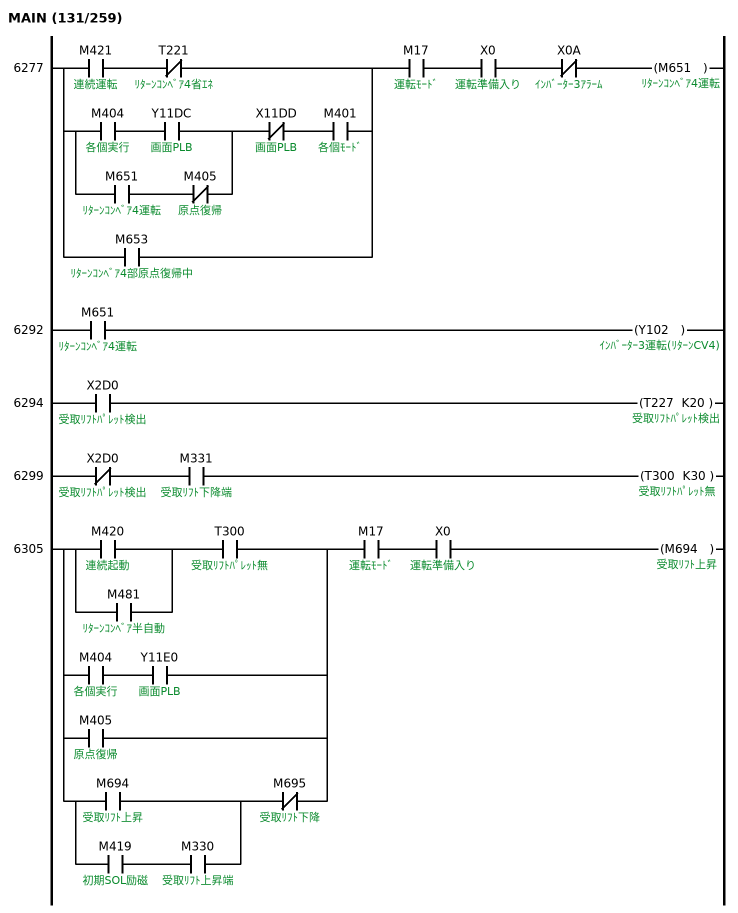
6277  LD      M421  ; 連続運転
      ANI     T221  ; ﾘﾀｰﾝｺﾝﾍﾞｱ4省ｴﾈ
      LD      M404  ; 各個実行
      AND     Y11DC  ; 画面PLB
      LD      M651  ; ﾘﾀｰﾝｺﾝﾍﾞｱ4運転
      ANI     M405  ; 原点復帰
      ORB
      ANI     X11DD  ; 画面PLB
      AND     M401  ; 各個ﾓｰﾄﾞ
      ORB
      OR      M653  ; ﾘﾀｰﾝｺﾝﾍﾞｱ4部原点復帰中
      AND     M17  ; 運転ﾓｰﾄﾞ
      AND     X0  ; 運転準備入り
      ANI     X0A  ; ｲﾝﾊﾞｰﾀｰ3ｱﾗｰﾑ
      OUT     M651  ; ﾘﾀｰﾝｺﾝﾍﾞｱ4運転
6292  LD      M651  ; ﾘﾀｰﾝｺﾝﾍﾞｱ4運転
      OUT     Y102  ; ｲﾝﾊﾞｰﾀｰ3運転(ﾘﾀｰﾝCV4)
6294  LD      X2D0  ; 受取ﾘﾌﾄﾊﾟﾚｯﾄ検出
      OUT     T227 K20  ; 受取ﾘﾌﾄﾊﾟﾚｯﾄ検出
6299  LDI     X2D0  ; 受取ﾘﾌﾄﾊﾟﾚｯﾄ検出
      AND     M331  ; 受取ﾘﾌﾄ下降端
      OUT     T300 K30  ; 受取ﾘﾌﾄﾊﾟﾚｯﾄ無
6305  LD      M420  ; 連続起動
      OR      M481  ; ﾘﾀｰﾝｺﾝﾍﾞｱ半自動
      AND     T300  ; 受取ﾘﾌﾄﾊﾟﾚｯﾄ無
      LD      M404  ; 各個実行
      AND     Y11E0  ; 画面PLB
      ORB
      OR      M405  ; 原点復帰
      LD      M694  ; 受取ﾘﾌﾄ上昇
      LD      M419  ; 初期SOL励磁
      AND     M330  ; 受取ﾘﾌﾄ上昇端
      ORB
      ANI     M695  ; 受取ﾘﾌﾄ下降
      ORB
      AND     M17  ; 運転ﾓｰﾄﾞ
      AND     X0  ; 運転準備入り
      OUT     M694  ; 受取ﾘﾌﾄ上昇
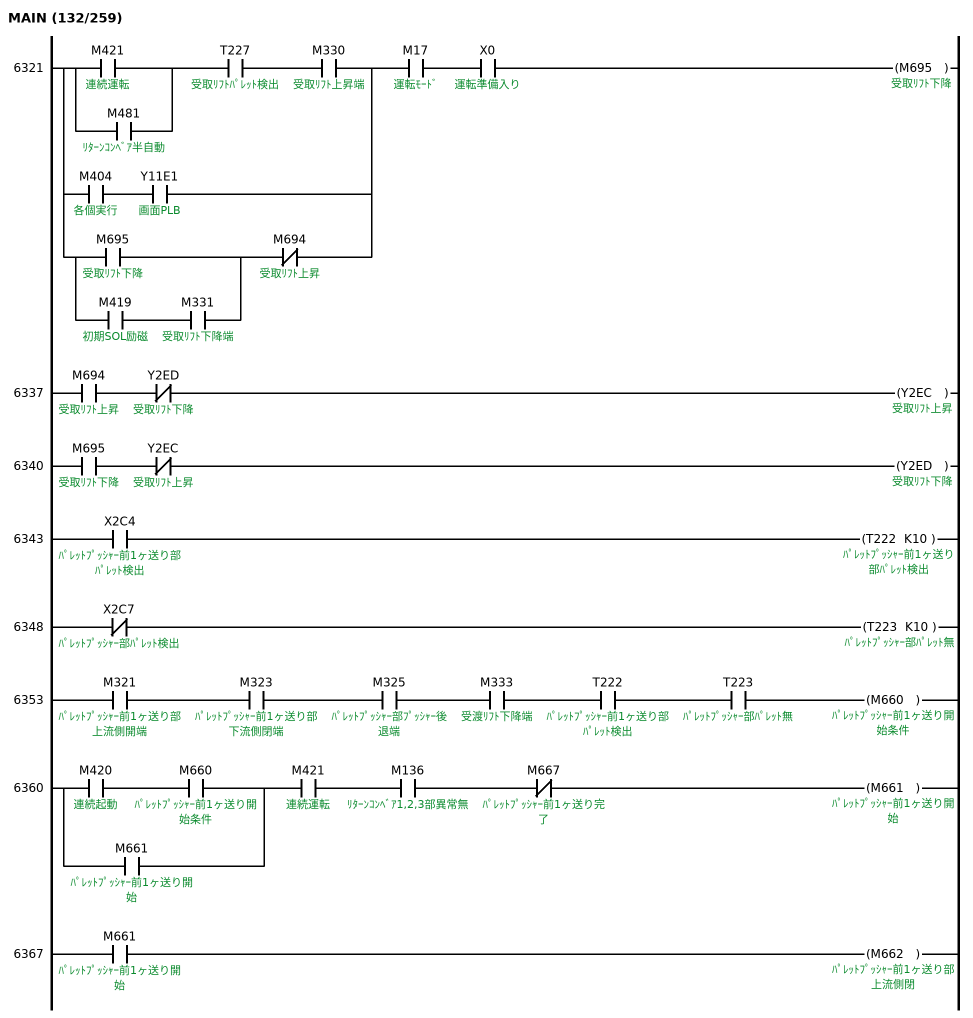
6321  LD      M421  ; 連続運転
      OR      M481  ; ﾘﾀｰﾝｺﾝﾍﾞｱ半自動
      AND     T227  ; 受取ﾘﾌﾄﾊﾟﾚｯﾄ検出
      AND     M330  ; 受取ﾘﾌﾄ上昇端
      LD      M404  ; 各個実行
      AND     Y11E1  ; 画面PLB
      ORB
      LD      M695  ; 受取ﾘﾌﾄ下降
      LD      M419  ; 初期SOL励磁
      AND     M331  ; 受取ﾘﾌﾄ下降端
      ORB
      ANI     M694  ; 受取ﾘﾌﾄ上昇
      ORB
      AND     M17  ; 運転ﾓｰﾄﾞ
      AND     X0  ; 運転準備入り
      OUT     M695  ; 受取ﾘﾌﾄ下降
6337  LD      M694  ; 受取ﾘﾌﾄ上昇
      ANI     Y2ED  ; 受取ﾘﾌﾄ下降
      OUT     Y2EC  ; 受取ﾘﾌﾄ上昇
6340  LD      M695  ; 受取ﾘﾌﾄ下降
      ANI     Y2EC  ; 受取ﾘﾌﾄ上昇
      OUT     Y2ED  ; 受取ﾘﾌﾄ下降
6343  LD      X2C4  ; ﾊﾟﾚｯﾄﾌﾟｯｼｬｰ前1ヶ送り部ﾊﾟﾚｯﾄ検出
      OUT     T222 K10  ; ﾊﾟﾚｯﾄﾌﾟｯｼｬｰ前1ヶ送り部ﾊﾟﾚｯﾄ検出
6348  LDI     X2C7  ; ﾊﾟﾚｯﾄﾌﾟｯｼｬｰ部ﾊﾟﾚｯﾄ検出
      OUT     T223 K10  ; ﾊﾟﾚｯﾄﾌﾟｯｼｬｰ部ﾊﾟﾚｯﾄ無
6353  LD      M321  ; ﾊﾟﾚｯﾄﾌﾟｯｼｬｰ前1ヶ送り部上流側開端
      AND     M323  ; ﾊﾟﾚｯﾄﾌﾟｯｼｬｰ前1ヶ送り部下流側閉端
      AND     M325  ; ﾊﾟﾚｯﾄﾌﾟｯｼｬｰ部ﾌﾟｯｼｬｰ後退端
      AND     M333  ; 受渡ﾘﾌﾄ下降端
      AND     T222  ; ﾊﾟﾚｯﾄﾌﾟｯｼｬｰ前1ヶ送り部ﾊﾟﾚｯﾄ検出
      AND     T223  ; ﾊﾟﾚｯﾄﾌﾟｯｼｬｰ部ﾊﾟﾚｯﾄ無
      OUT     M660  ; ﾊﾟﾚｯﾄﾌﾟｯｼｬｰ前1ヶ送り開始条件
6360  LD      M420  ; 連続起動
      AND     M660  ; ﾊﾟﾚｯﾄﾌﾟｯｼｬｰ前1ヶ送り開始条件
      OR      M661  ; ﾊﾟﾚｯﾄﾌﾟｯｼｬｰ前1ヶ送り開始
      AND     M421  ; 連続運転
      AND     M136  ; ﾘﾀｰﾝｺﾝﾍﾞｱ1,2,3部異常無
      ANI     M667  ; ﾊﾟﾚｯﾄﾌﾟｯｼｬｰ前1ヶ送り完了
      OUT     M661  ; ﾊﾟﾚｯﾄﾌﾟｯｼｬｰ前1ヶ送り開始
6367  LD      M661  ; ﾊﾟﾚｯﾄﾌﾟｯｼｬｰ前1ヶ送り開始
      OUT     M662  ; ﾊﾟﾚｯﾄﾌﾟｯｼｬｰ前1ヶ送り部上流側閉
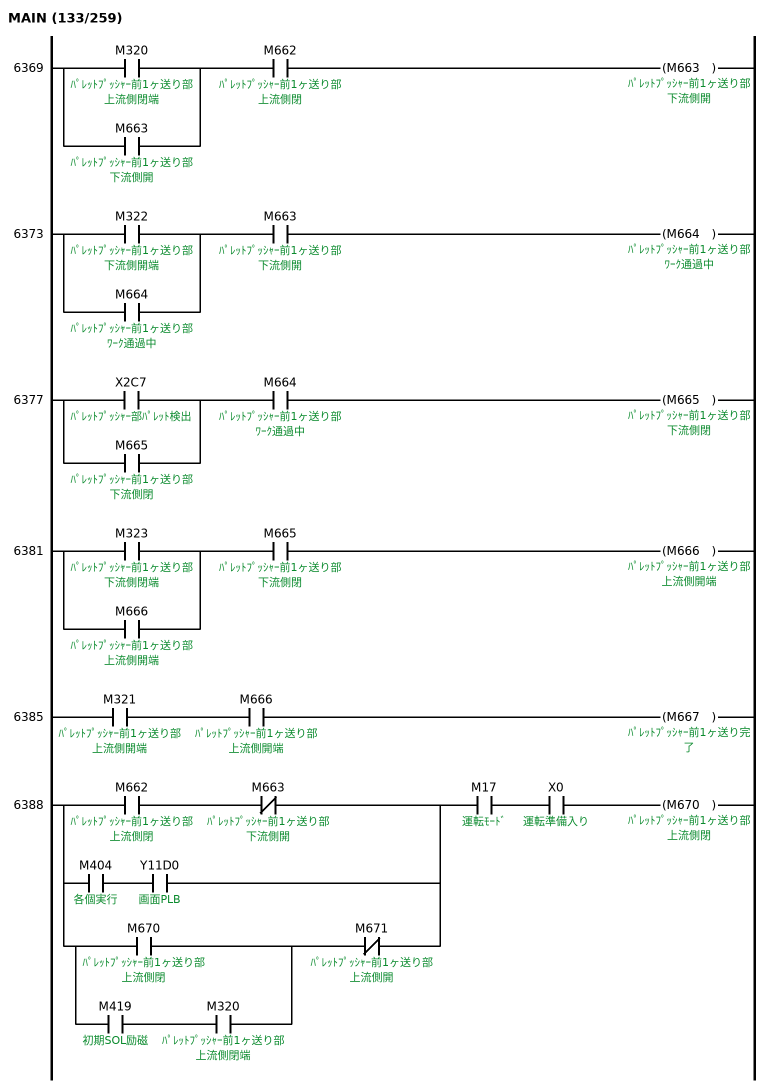
6369  LD      M320  ; ﾊﾟﾚｯﾄﾌﾟｯｼｬｰ前1ヶ送り部上流側閉端
      OR      M663  ; ﾊﾟﾚｯﾄﾌﾟｯｼｬｰ前1ヶ送り部下流側開
      AND     M662  ; ﾊﾟﾚｯﾄﾌﾟｯｼｬｰ前1ヶ送り部上流側閉
      OUT     M663  ; ﾊﾟﾚｯﾄﾌﾟｯｼｬｰ前1ヶ送り部下流側開
6373  LD      M322  ; ﾊﾟﾚｯﾄﾌﾟｯｼｬｰ前1ヶ送り部下流側開端
      OR      M664  ; ﾊﾟﾚｯﾄﾌﾟｯｼｬｰ前1ヶ送り部ﾜｰｸ通過中
      AND     M663  ; ﾊﾟﾚｯﾄﾌﾟｯｼｬｰ前1ヶ送り部下流側開
      OUT     M664  ; ﾊﾟﾚｯﾄﾌﾟｯｼｬｰ前1ヶ送り部ﾜｰｸ通過中
6377  LD      X2C7  ; ﾊﾟﾚｯﾄﾌﾟｯｼｬｰ部ﾊﾟﾚｯﾄ検出
      OR      M665  ; ﾊﾟﾚｯﾄﾌﾟｯｼｬｰ前1ヶ送り部下流側閉
      AND     M664  ; ﾊﾟﾚｯﾄﾌﾟｯｼｬｰ前1ヶ送り部ﾜｰｸ通過中
      OUT     M665  ; ﾊﾟﾚｯﾄﾌﾟｯｼｬｰ前1ヶ送り部下流側閉
6381  LD      M323  ; ﾊﾟﾚｯﾄﾌﾟｯｼｬｰ前1ヶ送り部下流側閉端
      OR      M666  ; ﾊﾟﾚｯﾄﾌﾟｯｼｬｰ前1ヶ送り部上流側開端
      AND     M665  ; ﾊﾟﾚｯﾄﾌﾟｯｼｬｰ前1ヶ送り部下流側閉
      OUT     M666  ; ﾊﾟﾚｯﾄﾌﾟｯｼｬｰ前1ヶ送り部上流側開端
6385  LD      M321  ; ﾊﾟﾚｯﾄﾌﾟｯｼｬｰ前1ヶ送り部上流側開端
      AND     M666  ; ﾊﾟﾚｯﾄﾌﾟｯｼｬｰ前1ヶ送り部上流側開端
      OUT     M667  ; ﾊﾟﾚｯﾄﾌﾟｯｼｬｰ前1ヶ送り完了
6388  LD      M662  ; ﾊﾟﾚｯﾄﾌﾟｯｼｬｰ前1ヶ送り部上流側閉
      ANI     M663  ; ﾊﾟﾚｯﾄﾌﾟｯｼｬｰ前1ヶ送り部下流側開
      LD      M404  ; 各個実行
      AND     Y11D0  ; 画面PLB
      ORB
      LD      M670  ; ﾊﾟﾚｯﾄﾌﾟｯｼｬｰ前1ヶ送り部上流側閉
      LD      M419  ; 初期SOL励磁
      AND     M320  ; ﾊﾟﾚｯﾄﾌﾟｯｼｬｰ前1ヶ送り部上流側閉端
      ORB
      ANI     M671  ; ﾊﾟﾚｯﾄﾌﾟｯｼｬｰ前1ヶ送り部上流側開
      ORB
      AND     M17  ; 運転ﾓｰﾄﾞ
      AND     X0  ; 運転準備入り
      OUT     M670  ; ﾊﾟﾚｯﾄﾌﾟｯｼｬｰ前1ヶ送り部上流側閉
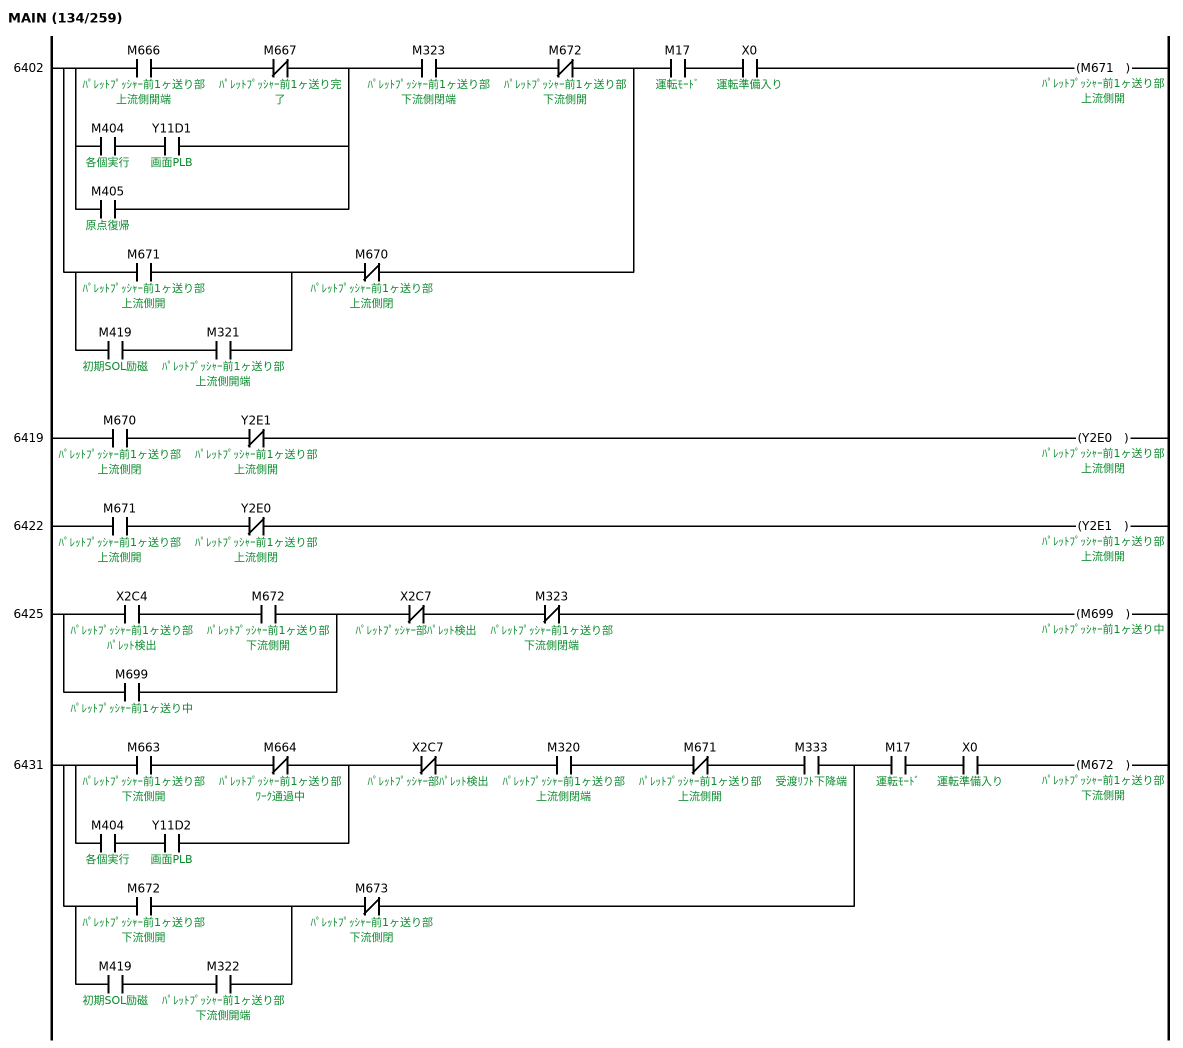
6402  LD      M666  ; ﾊﾟﾚｯﾄﾌﾟｯｼｬｰ前1ヶ送り部上流側開端
      ANI     M667  ; ﾊﾟﾚｯﾄﾌﾟｯｼｬｰ前1ヶ送り完了
      LD      M404  ; 各個実行
      AND     Y11D1  ; 画面PLB
      ORB
      OR      M405  ; 原点復帰
      AND     M323  ; ﾊﾟﾚｯﾄﾌﾟｯｼｬｰ前1ヶ送り部下流側閉端
      ANI     M672  ; ﾊﾟﾚｯﾄﾌﾟｯｼｬｰ前1ヶ送り部下流側開
      LD      M671  ; ﾊﾟﾚｯﾄﾌﾟｯｼｬｰ前1ヶ送り部上流側開
      LD      M419  ; 初期SOL励磁
      AND     M321  ; ﾊﾟﾚｯﾄﾌﾟｯｼｬｰ前1ヶ送り部上流側開端
      ORB
      ANI     M670  ; ﾊﾟﾚｯﾄﾌﾟｯｼｬｰ前1ヶ送り部上流側閉
      ORB
      AND     M17  ; 運転ﾓｰﾄﾞ
      AND     X0  ; 運転準備入り
      OUT     M671  ; ﾊﾟﾚｯﾄﾌﾟｯｼｬｰ前1ヶ送り部上流側開
6419  LD      M670  ; ﾊﾟﾚｯﾄﾌﾟｯｼｬｰ前1ヶ送り部上流側閉
      ANI     Y2E1  ; ﾊﾟﾚｯﾄﾌﾟｯｼｬｰ前1ヶ送り部上流側開
      OUT     Y2E0  ; ﾊﾟﾚｯﾄﾌﾟｯｼｬｰ前1ヶ送り部上流側閉
6422  LD      M671  ; ﾊﾟﾚｯﾄﾌﾟｯｼｬｰ前1ヶ送り部上流側開
      ANI     Y2E0  ; ﾊﾟﾚｯﾄﾌﾟｯｼｬｰ前1ヶ送り部上流側閉
      OUT     Y2E1  ; ﾊﾟﾚｯﾄﾌﾟｯｼｬｰ前1ヶ送り部上流側開
6425  LD      X2C4  ; ﾊﾟﾚｯﾄﾌﾟｯｼｬｰ前1ヶ送り部ﾊﾟﾚｯﾄ検出
      AND     M672  ; ﾊﾟﾚｯﾄﾌﾟｯｼｬｰ前1ヶ送り部下流側開
      OR      M699  ; ﾊﾟﾚｯﾄﾌﾟｯｼｬｰ前1ヶ送り中
      ANI     X2C7  ; ﾊﾟﾚｯﾄﾌﾟｯｼｬｰ部ﾊﾟﾚｯﾄ検出
      ANI     M323  ; ﾊﾟﾚｯﾄﾌﾟｯｼｬｰ前1ヶ送り部下流側閉端
      OUT     M699  ; ﾊﾟﾚｯﾄﾌﾟｯｼｬｰ前1ヶ送り中
6431  LD      M663  ; ﾊﾟﾚｯﾄﾌﾟｯｼｬｰ前1ヶ送り部下流側開
      ANI     M664  ; ﾊﾟﾚｯﾄﾌﾟｯｼｬｰ前1ヶ送り部ﾜｰｸ通過中
      LD      M404  ; 各個実行
      AND     Y11D2  ; 画面PLB
      ORB
      ANI     X2C7  ; ﾊﾟﾚｯﾄﾌﾟｯｼｬｰ部ﾊﾟﾚｯﾄ検出
      AND     M320  ; ﾊﾟﾚｯﾄﾌﾟｯｼｬｰ前1ヶ送り部上流側閉端
      ANI     M671  ; ﾊﾟﾚｯﾄﾌﾟｯｼｬｰ前1ヶ送り部上流側開
      AND     M333  ; 受渡ﾘﾌﾄ下降端
      LD      M672  ; ﾊﾟﾚｯﾄﾌﾟｯｼｬｰ前1ヶ送り部下流側開
      LD      M419  ; 初期SOL励磁
      AND     M322  ; ﾊﾟﾚｯﾄﾌﾟｯｼｬｰ前1ヶ送り部下流側開端
      ORB
      ANI     M673  ; ﾊﾟﾚｯﾄﾌﾟｯｼｬｰ前1ヶ送り部下流側閉
      ORB
      AND     M17  ; 運転ﾓｰﾄﾞ
      AND     X0  ; 運転準備入り
      OUT     M672  ; ﾊﾟﾚｯﾄﾌﾟｯｼｬｰ前1ヶ送り部下流側開
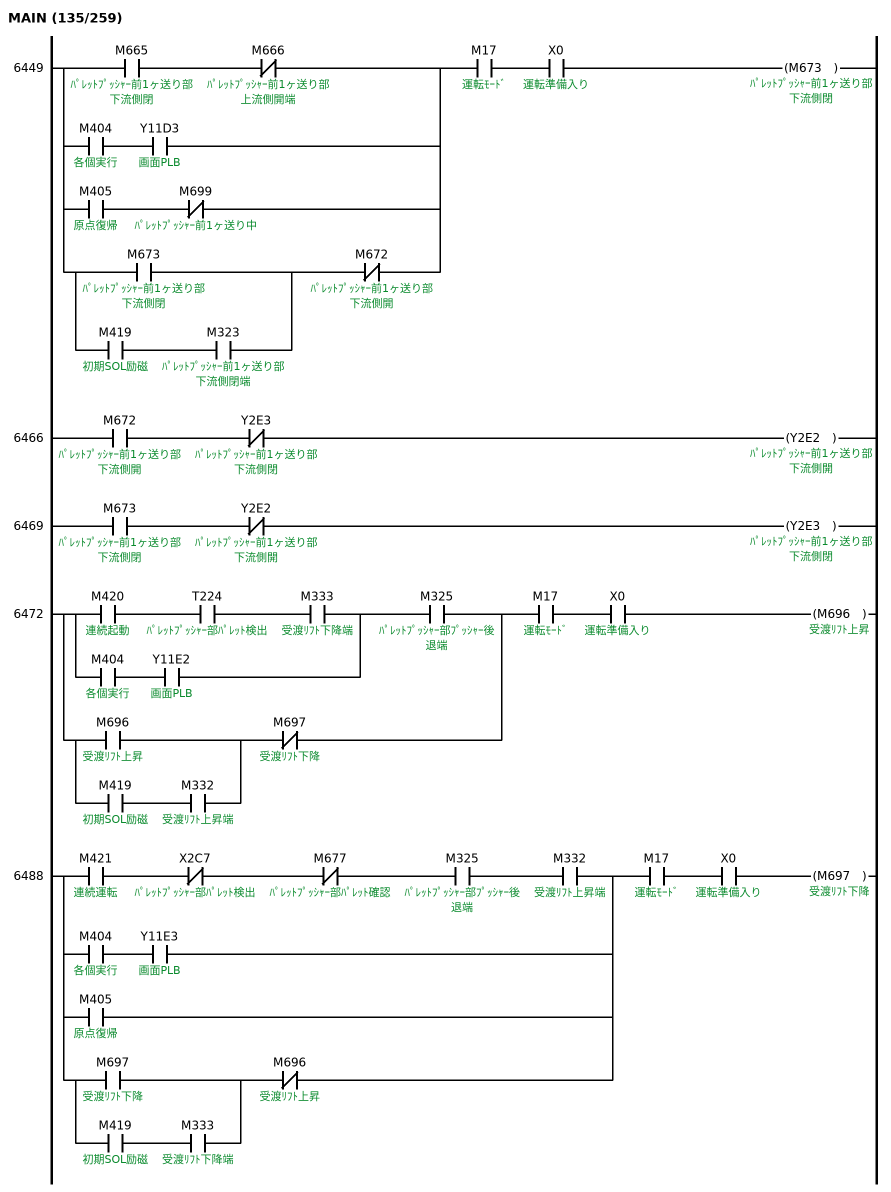
6449  LD      M665  ; ﾊﾟﾚｯﾄﾌﾟｯｼｬｰ前1ヶ送り部下流側閉
      ANI     M666  ; ﾊﾟﾚｯﾄﾌﾟｯｼｬｰ前1ヶ送り部上流側開端
      LD      M404  ; 各個実行
      AND     Y11D3  ; 画面PLB
      ORB
      LD      M405  ; 原点復帰
      ANI     M699  ; ﾊﾟﾚｯﾄﾌﾟｯｼｬｰ前1ヶ送り中
      ORB
      LD      M673  ; ﾊﾟﾚｯﾄﾌﾟｯｼｬｰ前1ヶ送り部下流側閉
      LD      M419  ; 初期SOL励磁
      AND     M323  ; ﾊﾟﾚｯﾄﾌﾟｯｼｬｰ前1ヶ送り部下流側閉端
      ORB
      ANI     M672  ; ﾊﾟﾚｯﾄﾌﾟｯｼｬｰ前1ヶ送り部下流側開
      ORB
      AND     M17  ; 運転ﾓｰﾄﾞ
      AND     X0  ; 運転準備入り
      OUT     M673  ; ﾊﾟﾚｯﾄﾌﾟｯｼｬｰ前1ヶ送り部下流側閉
6466  LD      M672  ; ﾊﾟﾚｯﾄﾌﾟｯｼｬｰ前1ヶ送り部下流側開
      ANI     Y2E3  ; ﾊﾟﾚｯﾄﾌﾟｯｼｬｰ前1ヶ送り部下流側閉
      OUT     Y2E2  ; ﾊﾟﾚｯﾄﾌﾟｯｼｬｰ前1ヶ送り部下流側開
6469  LD      M673  ; ﾊﾟﾚｯﾄﾌﾟｯｼｬｰ前1ヶ送り部下流側閉
      ANI     Y2E2  ; ﾊﾟﾚｯﾄﾌﾟｯｼｬｰ前1ヶ送り部下流側開
      OUT     Y2E3  ; ﾊﾟﾚｯﾄﾌﾟｯｼｬｰ前1ヶ送り部下流側閉
6472  LD      M420  ; 連続起動
      AND     T224  ; ﾊﾟﾚｯﾄﾌﾟｯｼｬｰ部ﾊﾟﾚｯﾄ検出
      AND     M333  ; 受渡ﾘﾌﾄ下降端
      LD      M404  ; 各個実行
      AND     Y11E2  ; 画面PLB
      ORB
      AND     M325  ; ﾊﾟﾚｯﾄﾌﾟｯｼｬｰ部ﾌﾟｯｼｬｰ後退端
      LD      M696  ; 受渡ﾘﾌﾄ上昇
      LD      M419  ; 初期SOL励磁
      AND     M332  ; 受渡ﾘﾌﾄ上昇端
      ORB
      ANI     M697  ; 受渡ﾘﾌﾄ下降
      ORB
      AND     M17  ; 運転ﾓｰﾄﾞ
      AND     X0  ; 運転準備入り
      OUT     M696  ; 受渡ﾘﾌﾄ上昇
6488  LD      M421  ; 連続運転
      ANI     X2C7  ; ﾊﾟﾚｯﾄﾌﾟｯｼｬｰ部ﾊﾟﾚｯﾄ検出
      ANI     M677  ; ﾊﾟﾚｯﾄﾌﾟｯｼｬｰ部ﾊﾟﾚｯﾄ確認
      AND     M325  ; ﾊﾟﾚｯﾄﾌﾟｯｼｬｰ部ﾌﾟｯｼｬｰ後退端
      AND     M332  ; 受渡ﾘﾌﾄ上昇端
      LD      M404  ; 各個実行
      AND     Y11E3  ; 画面PLB
      ORB
      OR      M405  ; 原点復帰
      LD      M697  ; 受渡ﾘﾌﾄ下降
      LD      M419  ; 初期SOL励磁
      AND     M333  ; 受渡ﾘﾌﾄ下降端
      ORB
      ANI     M696  ; 受渡ﾘﾌﾄ上昇
      ORB
      AND     M17  ; 運転ﾓｰﾄﾞ
      AND     X0  ; 運転準備入り
      OUT     M697  ; 受渡ﾘﾌﾄ下降
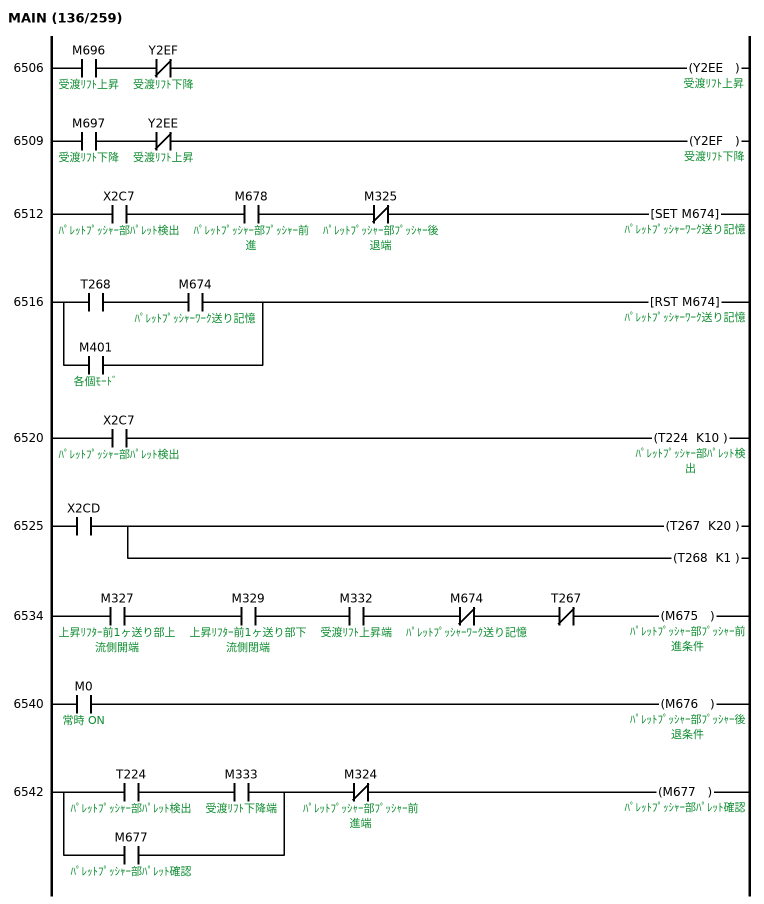
6506  LD      M696  ; 受渡ﾘﾌﾄ上昇
      ANI     Y2EF  ; 受渡ﾘﾌﾄ下降
      OUT     Y2EE  ; 受渡ﾘﾌﾄ上昇
6509  LD      M697  ; 受渡ﾘﾌﾄ下降
      ANI     Y2EE  ; 受渡ﾘﾌﾄ上昇
      OUT     Y2EF  ; 受渡ﾘﾌﾄ下降
6512  LD      X2C7  ; ﾊﾟﾚｯﾄﾌﾟｯｼｬｰ部ﾊﾟﾚｯﾄ検出
      AND     M678  ; ﾊﾟﾚｯﾄﾌﾟｯｼｬｰ部ﾌﾟｯｼｬｰ前進
      ANI     M325  ; ﾊﾟﾚｯﾄﾌﾟｯｼｬｰ部ﾌﾟｯｼｬｰ後退端
      SET     M674  ; ﾊﾟﾚｯﾄﾌﾟｯｼｬｰﾜｰｸ送り記憶
6516  LD      T268
      AND     M674  ; ﾊﾟﾚｯﾄﾌﾟｯｼｬｰﾜｰｸ送り記憶
      OR      M401  ; 各個ﾓｰﾄﾞ
      RST     M674  ; ﾊﾟﾚｯﾄﾌﾟｯｼｬｰﾜｰｸ送り記憶
6520  LD      X2C7  ; ﾊﾟﾚｯﾄﾌﾟｯｼｬｰ部ﾊﾟﾚｯﾄ検出
      OUT     T224 K10  ; ﾊﾟﾚｯﾄﾌﾟｯｼｬｰ部ﾊﾟﾚｯﾄ検出
6525  LD      X2CD
      OUT     T267 K20
      OUT     T268 K1
6534  LD      M327  ; 上昇ﾘﾌﾀｰ前1ヶ送り部上流側開端
      AND     M329  ; 上昇ﾘﾌﾀｰ前1ヶ送り部下流側閉端
      AND     M332  ; 受渡ﾘﾌﾄ上昇端
      ANI     M674  ; ﾊﾟﾚｯﾄﾌﾟｯｼｬｰﾜｰｸ送り記憶
      ANI     T267
      OUT     M675  ; ﾊﾟﾚｯﾄﾌﾟｯｼｬｰ部ﾌﾟｯｼｬｰ前進条件
6540  LD      M0  ; 常時 ON
      OUT     M676  ; ﾊﾟﾚｯﾄﾌﾟｯｼｬｰ部ﾌﾟｯｼｬｰ後退条件
6542  LD      T224  ; ﾊﾟﾚｯﾄﾌﾟｯｼｬｰ部ﾊﾟﾚｯﾄ検出
      AND     M333  ; 受渡ﾘﾌﾄ下降端
      OR      M677  ; ﾊﾟﾚｯﾄﾌﾟｯｼｬｰ部ﾊﾟﾚｯﾄ確認
      ANI     M324  ; ﾊﾟﾚｯﾄﾌﾟｯｼｬｰ部ﾌﾟｯｼｬｰ前進端
      OUT     M677  ; ﾊﾟﾚｯﾄﾌﾟｯｼｬｰ部ﾊﾟﾚｯﾄ確認
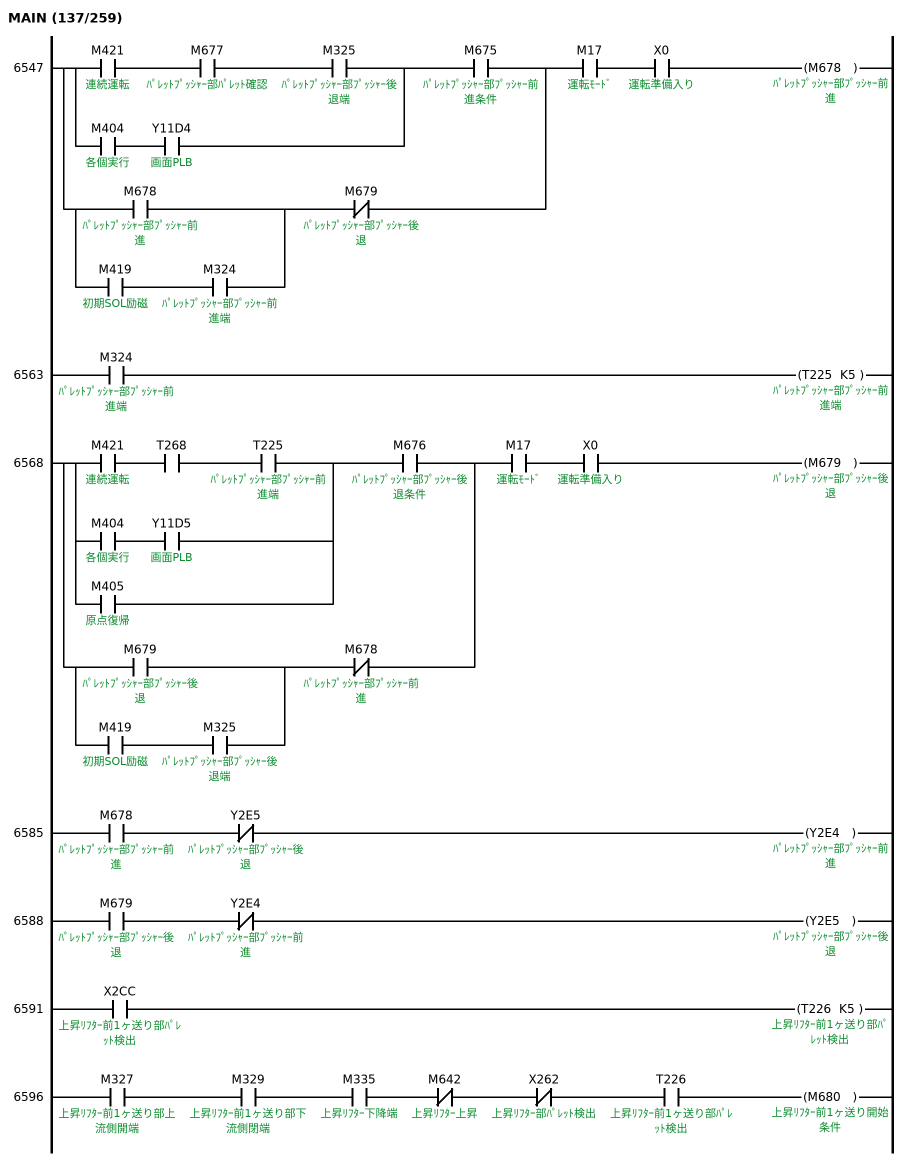
6547  LD      M421  ; 連続運転
      AND     M677  ; ﾊﾟﾚｯﾄﾌﾟｯｼｬｰ部ﾊﾟﾚｯﾄ確認
      AND     M325  ; ﾊﾟﾚｯﾄﾌﾟｯｼｬｰ部ﾌﾟｯｼｬｰ後退端
      LD      M404  ; 各個実行
      AND     Y11D4  ; 画面PLB
      ORB
      AND     M675  ; ﾊﾟﾚｯﾄﾌﾟｯｼｬｰ部ﾌﾟｯｼｬｰ前進条件
      LD      M678  ; ﾊﾟﾚｯﾄﾌﾟｯｼｬｰ部ﾌﾟｯｼｬｰ前進
      LD      M419  ; 初期SOL励磁
      AND     M324  ; ﾊﾟﾚｯﾄﾌﾟｯｼｬｰ部ﾌﾟｯｼｬｰ前進端
      ORB
      ANI     M679  ; ﾊﾟﾚｯﾄﾌﾟｯｼｬｰ部ﾌﾟｯｼｬｰ後退
      ORB
      AND     M17  ; 運転ﾓｰﾄﾞ
      AND     X0  ; 運転準備入り
      OUT     M678  ; ﾊﾟﾚｯﾄﾌﾟｯｼｬｰ部ﾌﾟｯｼｬｰ前進
6563  LD      M324  ; ﾊﾟﾚｯﾄﾌﾟｯｼｬｰ部ﾌﾟｯｼｬｰ前進端
      OUT     T225 K5  ; ﾊﾟﾚｯﾄﾌﾟｯｼｬｰ部ﾌﾟｯｼｬｰ前進端
6568  LD      M421  ; 連続運転
      AND     T268
      AND     T225  ; ﾊﾟﾚｯﾄﾌﾟｯｼｬｰ部ﾌﾟｯｼｬｰ前進端
      LD      M404  ; 各個実行
      AND     Y11D5  ; 画面PLB
      ORB
      OR      M405  ; 原点復帰
      AND     M676  ; ﾊﾟﾚｯﾄﾌﾟｯｼｬｰ部ﾌﾟｯｼｬｰ後退条件
      LD      M679  ; ﾊﾟﾚｯﾄﾌﾟｯｼｬｰ部ﾌﾟｯｼｬｰ後退
      LD      M419  ; 初期SOL励磁
      AND     M325  ; ﾊﾟﾚｯﾄﾌﾟｯｼｬｰ部ﾌﾟｯｼｬｰ後退端
      ORB
      ANI     M678  ; ﾊﾟﾚｯﾄﾌﾟｯｼｬｰ部ﾌﾟｯｼｬｰ前進
      ORB
      AND     M17  ; 運転ﾓｰﾄﾞ
      AND     X0  ; 運転準備入り
      OUT     M679  ; ﾊﾟﾚｯﾄﾌﾟｯｼｬｰ部ﾌﾟｯｼｬｰ後退
6585  LD      M678  ; ﾊﾟﾚｯﾄﾌﾟｯｼｬｰ部ﾌﾟｯｼｬｰ前進
      ANI     Y2E5  ; ﾊﾟﾚｯﾄﾌﾟｯｼｬｰ部ﾌﾟｯｼｬｰ後退
      OUT     Y2E4  ; ﾊﾟﾚｯﾄﾌﾟｯｼｬｰ部ﾌﾟｯｼｬｰ前進
6588  LD      M679  ; ﾊﾟﾚｯﾄﾌﾟｯｼｬｰ部ﾌﾟｯｼｬｰ後退
      ANI     Y2E4  ; ﾊﾟﾚｯﾄﾌﾟｯｼｬｰ部ﾌﾟｯｼｬｰ前進
      OUT     Y2E5  ; ﾊﾟﾚｯﾄﾌﾟｯｼｬｰ部ﾌﾟｯｼｬｰ後退
6591  LD      X2CC  ; 上昇ﾘﾌﾀｰ前1ヶ送り部ﾊﾟﾚｯﾄ検出
      OUT     T226 K5  ; 上昇ﾘﾌﾀｰ前1ヶ送り部ﾊﾟﾚｯﾄ検出
6596  LD      M327  ; 上昇ﾘﾌﾀｰ前1ヶ送り部上流側開端
      AND     M329  ; 上昇ﾘﾌﾀｰ前1ヶ送り部下流側閉端
      AND     M335  ; 上昇ﾘﾌﾀｰ下降端
      ANI     M642  ; 上昇ﾘﾌﾀｰ上昇
      ANI     X262  ; 上昇ﾘﾌﾀｰ部ﾊﾟﾚｯﾄ検出
      AND     T226  ; 上昇ﾘﾌﾀｰ前1ヶ送り部ﾊﾟﾚｯﾄ検出
      OUT     M680  ; 上昇ﾘﾌﾀｰ前1ヶ送り開始条件
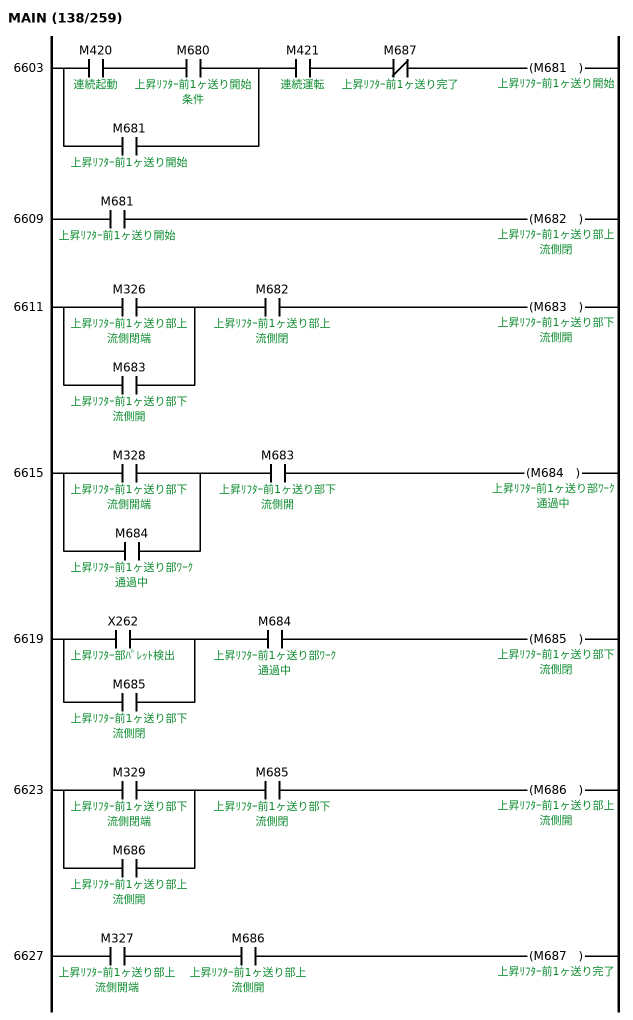
6603  LD      M420  ; 連続起動
      AND     M680  ; 上昇ﾘﾌﾀｰ前1ヶ送り開始条件
      OR      M681  ; 上昇ﾘﾌﾀｰ前1ヶ送り開始
      AND     M421  ; 連続運転
      ANI     M687  ; 上昇ﾘﾌﾀｰ前1ヶ送り完了
      OUT     M681  ; 上昇ﾘﾌﾀｰ前1ヶ送り開始
6609  LD      M681  ; 上昇ﾘﾌﾀｰ前1ヶ送り開始
      OUT     M682  ; 上昇ﾘﾌﾀｰ前1ヶ送り部上流側閉
6611  LD      M326  ; 上昇ﾘﾌﾀｰ前1ヶ送り部上流側閉端
      OR      M683  ; 上昇ﾘﾌﾀｰ前1ヶ送り部下流側開
      AND     M682  ; 上昇ﾘﾌﾀｰ前1ヶ送り部上流側閉
      OUT     M683  ; 上昇ﾘﾌﾀｰ前1ヶ送り部下流側開
6615  LD      M328  ; 上昇ﾘﾌﾀｰ前1ヶ送り部下流側開端
      OR      M684  ; 上昇ﾘﾌﾀｰ前1ヶ送り部ﾜｰｸ通過中
      AND     M683  ; 上昇ﾘﾌﾀｰ前1ヶ送り部下流側開
      OUT     M684  ; 上昇ﾘﾌﾀｰ前1ヶ送り部ﾜｰｸ通過中
6619  LD      X262  ; 上昇ﾘﾌﾀｰ部ﾊﾟﾚｯﾄ検出
      OR      M685  ; 上昇ﾘﾌﾀｰ前1ヶ送り部下流側閉
      AND     M684  ; 上昇ﾘﾌﾀｰ前1ヶ送り部ﾜｰｸ通過中
      OUT     M685  ; 上昇ﾘﾌﾀｰ前1ヶ送り部下流側閉
6623  LD      M329  ; 上昇ﾘﾌﾀｰ前1ヶ送り部下流側閉端
      OR      M686  ; 上昇ﾘﾌﾀｰ前1ヶ送り部上流側開
      AND     M685  ; 上昇ﾘﾌﾀｰ前1ヶ送り部下流側閉
      OUT     M686  ; 上昇ﾘﾌﾀｰ前1ヶ送り部上流側開
6627  LD      M327  ; 上昇ﾘﾌﾀｰ前1ヶ送り部上流側開端
      AND     M686  ; 上昇ﾘﾌﾀｰ前1ヶ送り部上流側開
      OUT     M687  ; 上昇ﾘﾌﾀｰ前1ヶ送り完了
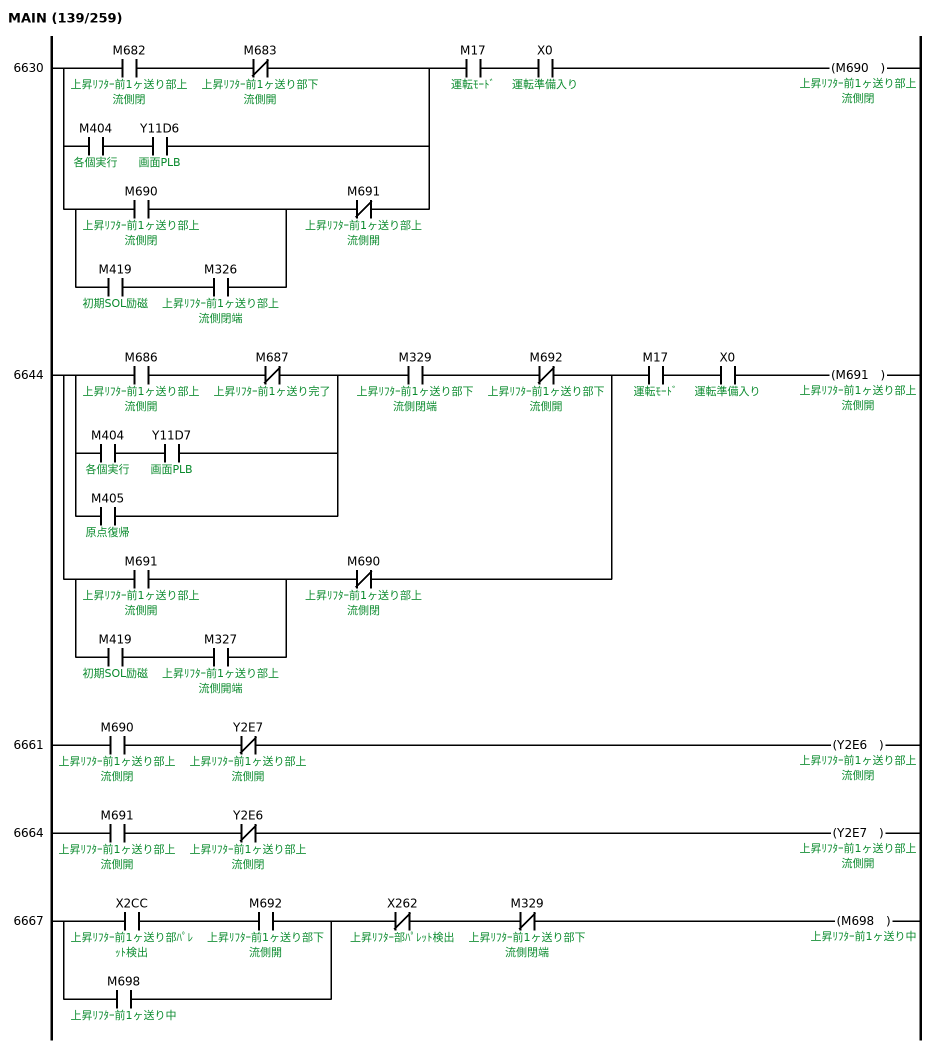
6630  LD      M682  ; 上昇ﾘﾌﾀｰ前1ヶ送り部上流側閉
      ANI     M683  ; 上昇ﾘﾌﾀｰ前1ヶ送り部下流側開
      LD      M404  ; 各個実行
      AND     Y11D6  ; 画面PLB
      ORB
      LD      M690  ; 上昇ﾘﾌﾀｰ前1ヶ送り部上流側閉
      LD      M419  ; 初期SOL励磁
      AND     M326  ; 上昇ﾘﾌﾀｰ前1ヶ送り部上流側閉端
      ORB
      ANI     M691  ; 上昇ﾘﾌﾀｰ前1ヶ送り部上流側開
      ORB
      AND     M17  ; 運転ﾓｰﾄﾞ
      AND     X0  ; 運転準備入り
      OUT     M690  ; 上昇ﾘﾌﾀｰ前1ヶ送り部上流側閉
6644  LD      M686  ; 上昇ﾘﾌﾀｰ前1ヶ送り部上流側開
      ANI     M687  ; 上昇ﾘﾌﾀｰ前1ヶ送り完了
      LD      M404  ; 各個実行
      AND     Y11D7  ; 画面PLB
      ORB
      OR      M405  ; 原点復帰
      AND     M329  ; 上昇ﾘﾌﾀｰ前1ヶ送り部下流側閉端
      ANI     M692  ; 上昇ﾘﾌﾀｰ前1ヶ送り部下流側開
      LD      M691  ; 上昇ﾘﾌﾀｰ前1ヶ送り部上流側開
      LD      M419  ; 初期SOL励磁
      AND     M327  ; 上昇ﾘﾌﾀｰ前1ヶ送り部上流側開端
      ORB
      ANI     M690  ; 上昇ﾘﾌﾀｰ前1ヶ送り部上流側閉
      ORB
      AND     M17  ; 運転ﾓｰﾄﾞ
      AND     X0  ; 運転準備入り
      OUT     M691  ; 上昇ﾘﾌﾀｰ前1ヶ送り部上流側開
6661  LD      M690  ; 上昇ﾘﾌﾀｰ前1ヶ送り部上流側閉
      ANI     Y2E7  ; 上昇ﾘﾌﾀｰ前1ヶ送り部上流側開
      OUT     Y2E6  ; 上昇ﾘﾌﾀｰ前1ヶ送り部上流側閉
6664  LD      M691  ; 上昇ﾘﾌﾀｰ前1ヶ送り部上流側開
      ANI     Y2E6  ; 上昇ﾘﾌﾀｰ前1ヶ送り部上流側閉
      OUT     Y2E7  ; 上昇ﾘﾌﾀｰ前1ヶ送り部上流側開
6667  LD      X2CC  ; 上昇ﾘﾌﾀｰ前1ヶ送り部ﾊﾟﾚｯﾄ検出
      AND     M692  ; 上昇ﾘﾌﾀｰ前1ヶ送り部下流側開
      OR      M698  ; 上昇ﾘﾌﾀｰ前1ヶ送り中
      ANI     X262  ; 上昇ﾘﾌﾀｰ部ﾊﾟﾚｯﾄ検出
      ANI     M329  ; 上昇ﾘﾌﾀｰ前1ヶ送り部下流側閉端
      OUT     M698  ; 上昇ﾘﾌﾀｰ前1ヶ送り中
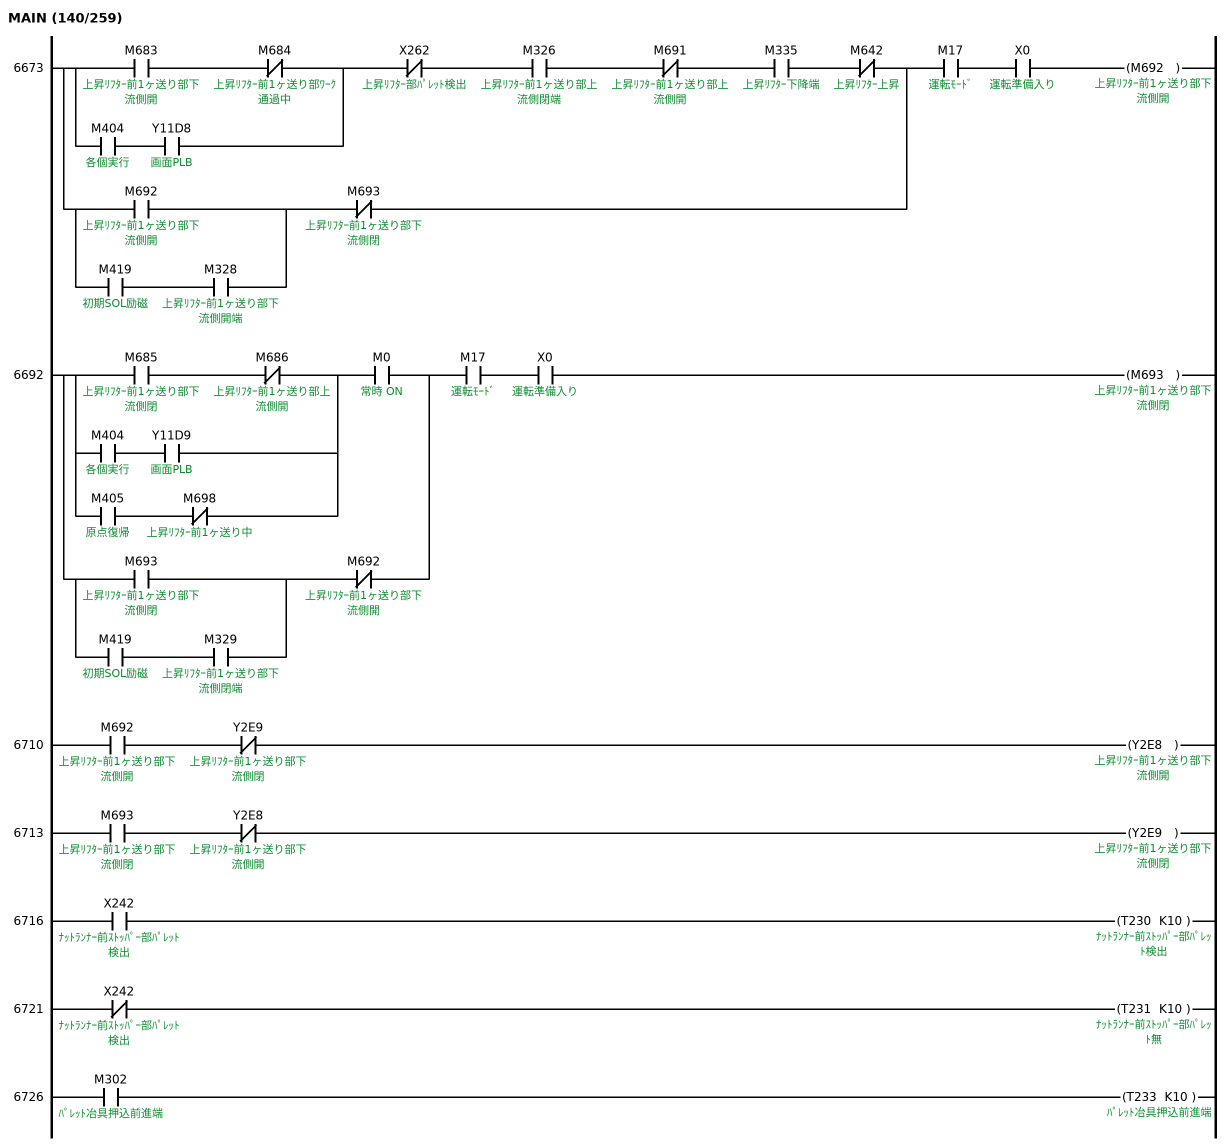
6673  LD      M683  ; 上昇ﾘﾌﾀｰ前1ヶ送り部下流側開
      ANI     M684  ; 上昇ﾘﾌﾀｰ前1ヶ送り部ﾜｰｸ通過中
      LD      M404  ; 各個実行
      AND     Y11D8  ; 画面PLB
      ORB
      ANI     X262  ; 上昇ﾘﾌﾀｰ部ﾊﾟﾚｯﾄ検出
      AND     M326  ; 上昇ﾘﾌﾀｰ前1ヶ送り部上流側閉端
      ANI     M691  ; 上昇ﾘﾌﾀｰ前1ヶ送り部上流側開
      AND     M335  ; 上昇ﾘﾌﾀｰ下降端
      ANI     M642  ; 上昇ﾘﾌﾀｰ上昇
      LD      M692  ; 上昇ﾘﾌﾀｰ前1ヶ送り部下流側開
      LD      M419  ; 初期SOL励磁
      AND     M328  ; 上昇ﾘﾌﾀｰ前1ヶ送り部下流側開端
      ORB
      ANI     M693  ; 上昇ﾘﾌﾀｰ前1ヶ送り部下流側閉
      ORB
      AND     M17  ; 運転ﾓｰﾄﾞ
      AND     X0  ; 運転準備入り
      OUT     M692  ; 上昇ﾘﾌﾀｰ前1ヶ送り部下流側開
6692  LD      M685  ; 上昇ﾘﾌﾀｰ前1ヶ送り部下流側閉
      ANI     M686  ; 上昇ﾘﾌﾀｰ前1ヶ送り部上流側開
      LD      M404  ; 各個実行
      AND     Y11D9  ; 画面PLB
      ORB
      LD      M405  ; 原点復帰
      ANI     M698  ; 上昇ﾘﾌﾀｰ前1ヶ送り中
      ORB
      AND     M0  ; 常時 ON
      LD      M693  ; 上昇ﾘﾌﾀｰ前1ヶ送り部下流側閉
      LD      M419  ; 初期SOL励磁
      AND     M329  ; 上昇ﾘﾌﾀｰ前1ヶ送り部下流側閉端
      ORB
      ANI     M692  ; 上昇ﾘﾌﾀｰ前1ヶ送り部下流側開
      ORB
      AND     M17  ; 運転ﾓｰﾄﾞ
      AND     X0  ; 運転準備入り
      OUT     M693  ; 上昇ﾘﾌﾀｰ前1ヶ送り部下流側閉
6710  LD      M692  ; 上昇ﾘﾌﾀｰ前1ヶ送り部下流側開
      ANI     Y2E9  ; 上昇ﾘﾌﾀｰ前1ヶ送り部下流側閉
      OUT     Y2E8  ; 上昇ﾘﾌﾀｰ前1ヶ送り部下流側開
6713  LD      M693  ; 上昇ﾘﾌﾀｰ前1ヶ送り部下流側閉
      ANI     Y2E8  ; 上昇ﾘﾌﾀｰ前1ヶ送り部下流側開
      OUT     Y2E9  ; 上昇ﾘﾌﾀｰ前1ヶ送り部下流側閉
6716  LD      X242  ; ﾅｯﾄﾗﾝﾅｰ前ｽﾄｯﾊﾟｰ部ﾊﾟﾚｯﾄ検出
      OUT     T230 K10  ; ﾅｯﾄﾗﾝﾅｰ前ｽﾄｯﾊﾟｰ部ﾊﾟﾚｯﾄ検出
6721  LDI     X242  ; ﾅｯﾄﾗﾝﾅｰ前ｽﾄｯﾊﾟｰ部ﾊﾟﾚｯﾄ検出
      OUT     T231 K10  ; ﾅｯﾄﾗﾝﾅｰ前ｽﾄｯﾊﾟｰ部ﾊﾟﾚｯﾄ無
6726  LD      M302  ; ﾊﾟﾚｯﾄ冶具押込前進端
      OUT     T233 K10  ; ﾊﾟﾚｯﾄ冶具押込前進端
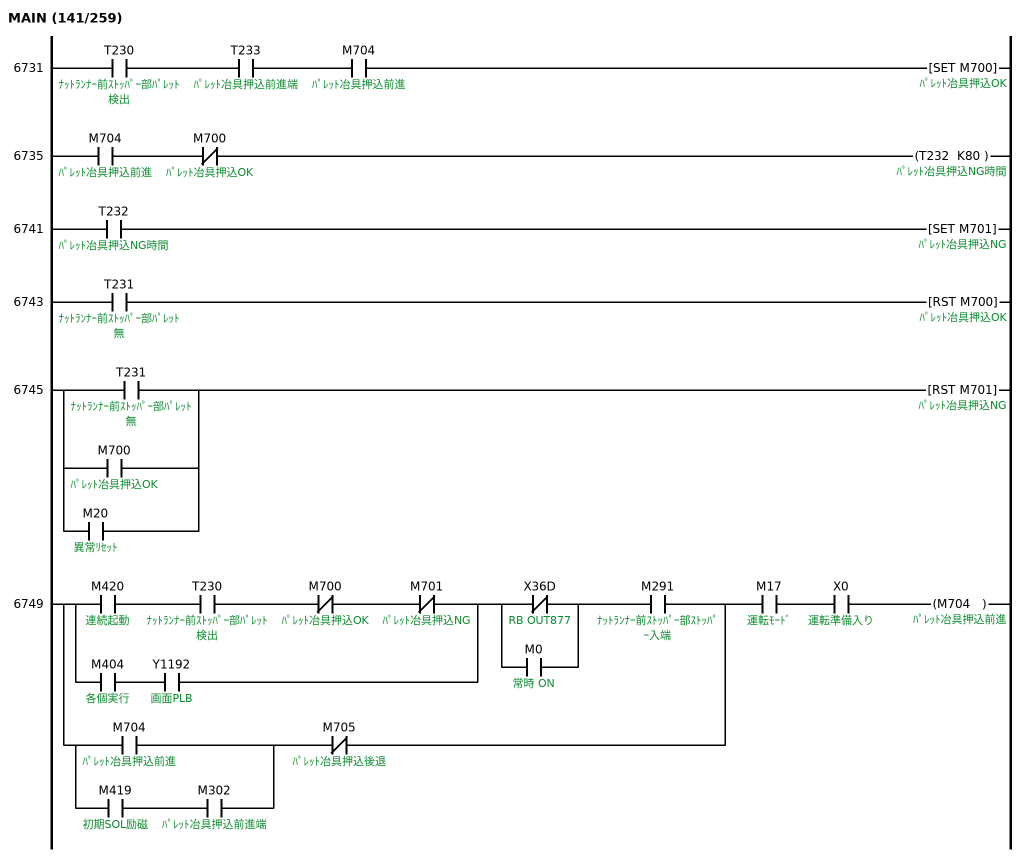
6731  LD      T230  ; ﾅｯﾄﾗﾝﾅｰ前ｽﾄｯﾊﾟｰ部ﾊﾟﾚｯﾄ検出
      AND     T233  ; ﾊﾟﾚｯﾄ冶具押込前進端
      AND     M704  ; ﾊﾟﾚｯﾄ冶具押込前進
      SET     M700  ; ﾊﾟﾚｯﾄ冶具押込OK
6735  LD      M704  ; ﾊﾟﾚｯﾄ冶具押込前進
      ANI     M700  ; ﾊﾟﾚｯﾄ冶具押込OK
      OUT     T232 K80  ; ﾊﾟﾚｯﾄ冶具押込NG時間
6741  LD      T232  ; ﾊﾟﾚｯﾄ冶具押込NG時間
      SET     M701  ; ﾊﾟﾚｯﾄ冶具押込NG
6743  LD      T231  ; ﾅｯﾄﾗﾝﾅｰ前ｽﾄｯﾊﾟｰ部ﾊﾟﾚｯﾄ無
      RST     M700  ; ﾊﾟﾚｯﾄ冶具押込OK
6745  LD      T231  ; ﾅｯﾄﾗﾝﾅｰ前ｽﾄｯﾊﾟｰ部ﾊﾟﾚｯﾄ無
      OR      M700  ; ﾊﾟﾚｯﾄ冶具押込OK
      OR      M20  ; 異常ﾘｾｯﾄ
      RST     M701  ; ﾊﾟﾚｯﾄ冶具押込NG
6749  LD      M420  ; 連続起動
      AND     T230  ; ﾅｯﾄﾗﾝﾅｰ前ｽﾄｯﾊﾟｰ部ﾊﾟﾚｯﾄ検出
      ANI     M700  ; ﾊﾟﾚｯﾄ冶具押込OK
      ANI     M701  ; ﾊﾟﾚｯﾄ冶具押込NG
      LD      M404  ; 各個実行
      AND     Y1192  ; 画面PLB
      ORB
      LDI     X36D  ; RB OUT877
      OR      M0  ; 常時 ON
      ANB
      AND     M291  ; ﾅｯﾄﾗﾝﾅｰ前ｽﾄｯﾊﾟｰ部ｽﾄｯﾊﾟｰ入端
      LD      M704  ; ﾊﾟﾚｯﾄ冶具押込前進
      LD      M419  ; 初期SOL励磁
      AND     M302  ; ﾊﾟﾚｯﾄ冶具押込前進端
      ORB
      ANI     M705  ; ﾊﾟﾚｯﾄ冶具押込後退
      ORB
      AND     M17  ; 運転ﾓｰﾄﾞ
      AND     X0  ; 運転準備入り
      OUT     M704  ; ﾊﾟﾚｯﾄ冶具押込前進
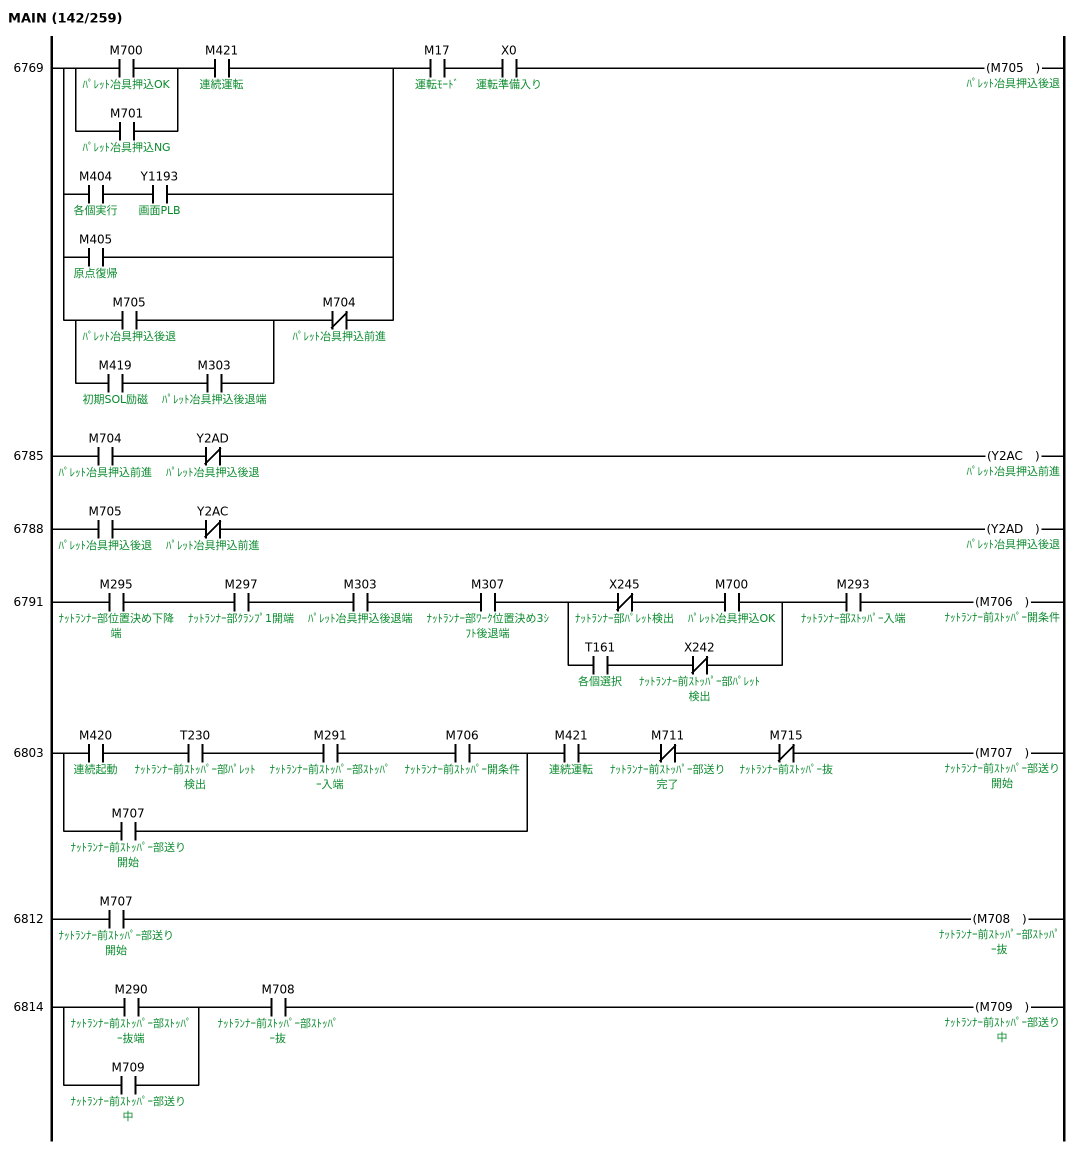
6769  LD      M700  ; ﾊﾟﾚｯﾄ冶具押込OK
      OR      M701  ; ﾊﾟﾚｯﾄ冶具押込NG
      AND     M421  ; 連続運転
      LD      M404  ; 各個実行
      AND     Y1193  ; 画面PLB
      ORB
      OR      M405  ; 原点復帰
      LD      M705  ; ﾊﾟﾚｯﾄ冶具押込後退
      LD      M419  ; 初期SOL励磁
      AND     M303  ; ﾊﾟﾚｯﾄ冶具押込後退端
      ORB
      ANI     M704  ; ﾊﾟﾚｯﾄ冶具押込前進
      ORB
      AND     M17  ; 運転ﾓｰﾄﾞ
      AND     X0  ; 運転準備入り
      OUT     M705  ; ﾊﾟﾚｯﾄ冶具押込後退
6785  LD      M704  ; ﾊﾟﾚｯﾄ冶具押込前進
      ANI     Y2AD  ; ﾊﾟﾚｯﾄ冶具押込後退
      OUT     Y2AC  ; ﾊﾟﾚｯﾄ冶具押込前進
6788  LD      M705  ; ﾊﾟﾚｯﾄ冶具押込後退
      ANI     Y2AC  ; ﾊﾟﾚｯﾄ冶具押込前進
      OUT     Y2AD  ; ﾊﾟﾚｯﾄ冶具押込後退
6791  LD      M295  ; ﾅｯﾄﾗﾝﾅｰ部位置決め下降端
      AND     M297  ; ﾅｯﾄﾗﾝﾅｰ部ｸﾗﾝﾌﾟ1開端
      AND     M303  ; ﾊﾟﾚｯﾄ冶具押込後退端
      AND     M307  ; ﾅｯﾄﾗﾝﾅｰ部ﾜｰｸ位置決め3ｼﾌﾄ後退端
      LDI     X245  ; ﾅｯﾄﾗﾝﾅｰ部ﾊﾟﾚｯﾄ検出
      AND     M700  ; ﾊﾟﾚｯﾄ冶具押込OK
      LD      T161  ; 各個選択
      ANI     X242  ; ﾅｯﾄﾗﾝﾅｰ前ｽﾄｯﾊﾟｰ部ﾊﾟﾚｯﾄ検出
      ORB
      ANB
      AND     M293  ; ﾅｯﾄﾗﾝﾅｰ部ｽﾄｯﾊﾟｰ入端
      OUT     M706  ; ﾅｯﾄﾗﾝﾅｰ前ｽﾄｯﾊﾟｰ開条件
6803  LD      M420  ; 連続起動
      AND     T230  ; ﾅｯﾄﾗﾝﾅｰ前ｽﾄｯﾊﾟｰ部ﾊﾟﾚｯﾄ検出
      AND     M291  ; ﾅｯﾄﾗﾝﾅｰ前ｽﾄｯﾊﾟｰ部ｽﾄｯﾊﾟｰ入端
      AND     M706  ; ﾅｯﾄﾗﾝﾅｰ前ｽﾄｯﾊﾟｰ開条件
      OR      M707  ; ﾅｯﾄﾗﾝﾅｰ前ｽﾄｯﾊﾟｰ部送り開始
      AND     M421  ; 連続運転
      ANI     M711  ; ﾅｯﾄﾗﾝﾅｰ前ｽﾄｯﾊﾟｰ部送り完了
      ANI     M715  ; ﾅｯﾄﾗﾝﾅｰ前ｽﾄｯﾊﾟｰ抜
      OUT     M707  ; ﾅｯﾄﾗﾝﾅｰ前ｽﾄｯﾊﾟｰ部送り開始
6812  LD      M707  ; ﾅｯﾄﾗﾝﾅｰ前ｽﾄｯﾊﾟｰ部送り開始
      OUT     M708  ; ﾅｯﾄﾗﾝﾅｰ前ｽﾄｯﾊﾟｰ部ｽﾄｯﾊﾟｰ抜
6814  LD      M290  ; ﾅｯﾄﾗﾝﾅｰ前ｽﾄｯﾊﾟｰ部ｽﾄｯﾊﾟｰ抜端
      OR      M709  ; ﾅｯﾄﾗﾝﾅｰ前ｽﾄｯﾊﾟｰ部送り中
      AND     M708  ; ﾅｯﾄﾗﾝﾅｰ前ｽﾄｯﾊﾟｰ部ｽﾄｯﾊﾟｰ抜
      OUT     M709  ; ﾅｯﾄﾗﾝﾅｰ前ｽﾄｯﾊﾟｰ部送り中
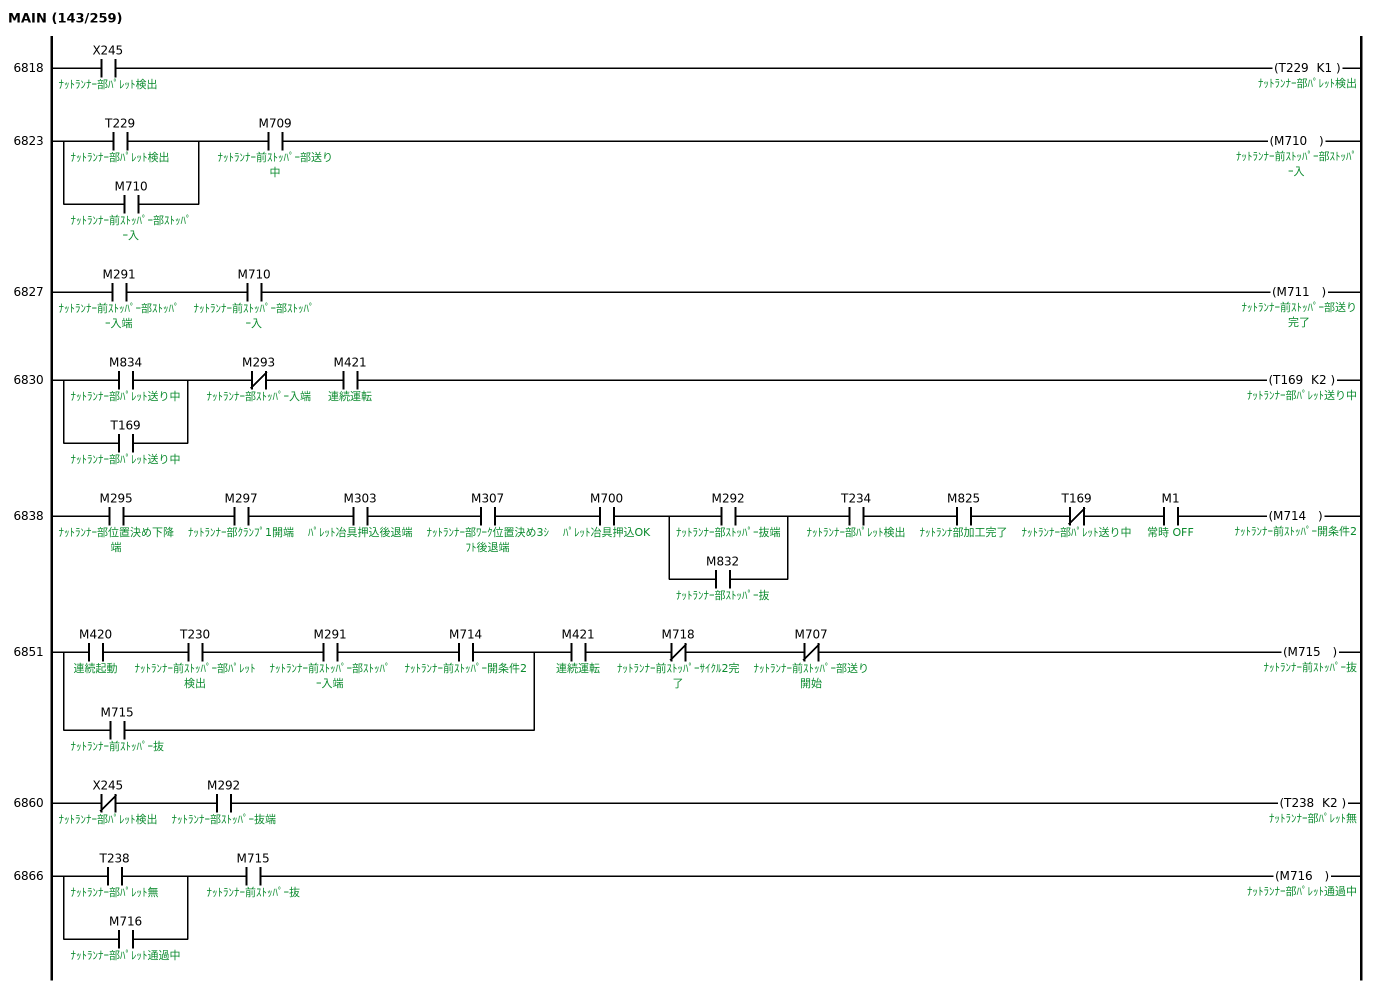
6818  LD      X245  ; ﾅｯﾄﾗﾝﾅｰ部ﾊﾟﾚｯﾄ検出
      OUT     T229 K1  ; ﾅｯﾄﾗﾝﾅｰ部ﾊﾟﾚｯﾄ検出
6823  LD      T229  ; ﾅｯﾄﾗﾝﾅｰ部ﾊﾟﾚｯﾄ検出
      OR      M710  ; ﾅｯﾄﾗﾝﾅｰ前ｽﾄｯﾊﾟｰ部ｽﾄｯﾊﾟｰ入
      AND     M709  ; ﾅｯﾄﾗﾝﾅｰ前ｽﾄｯﾊﾟｰ部送り中
      OUT     M710  ; ﾅｯﾄﾗﾝﾅｰ前ｽﾄｯﾊﾟｰ部ｽﾄｯﾊﾟｰ入
6827  LD      M291  ; ﾅｯﾄﾗﾝﾅｰ前ｽﾄｯﾊﾟｰ部ｽﾄｯﾊﾟｰ入端
      AND     M710  ; ﾅｯﾄﾗﾝﾅｰ前ｽﾄｯﾊﾟｰ部ｽﾄｯﾊﾟｰ入
      OUT     M711  ; ﾅｯﾄﾗﾝﾅｰ前ｽﾄｯﾊﾟｰ部送り完了
6830  LD      M834  ; ﾅｯﾄﾗﾝﾅｰ部ﾊﾟﾚｯﾄ送り中
      OR      T169  ; ﾅｯﾄﾗﾝﾅｰ部ﾊﾟﾚｯﾄ送り中
      ANI     M293  ; ﾅｯﾄﾗﾝﾅｰ部ｽﾄｯﾊﾟｰ入端
      AND     M421  ; 連続運転
      OUT     T169 K2  ; ﾅｯﾄﾗﾝﾅｰ部ﾊﾟﾚｯﾄ送り中
6838  LD      M295  ; ﾅｯﾄﾗﾝﾅｰ部位置決め下降端
      AND     M297  ; ﾅｯﾄﾗﾝﾅｰ部ｸﾗﾝﾌﾟ1開端
      AND     M303  ; ﾊﾟﾚｯﾄ冶具押込後退端
      AND     M307  ; ﾅｯﾄﾗﾝﾅｰ部ﾜｰｸ位置決め3ｼﾌﾄ後退端
      AND     M700  ; ﾊﾟﾚｯﾄ冶具押込OK
      LD      M292  ; ﾅｯﾄﾗﾝﾅｰ部ｽﾄｯﾊﾟｰ抜端
      OR      M832  ; ﾅｯﾄﾗﾝﾅｰ部ｽﾄｯﾊﾟｰ抜
      ANB
      AND     T234  ; ﾅｯﾄﾗﾝﾅｰ部ﾊﾟﾚｯﾄ検出
      AND     M825  ; ﾅｯﾄﾗﾝﾅ部加工完了
      ANI     T169  ; ﾅｯﾄﾗﾝﾅｰ部ﾊﾟﾚｯﾄ送り中
      AND     M1  ; 常時 OFF
      OUT     M714  ; ﾅｯﾄﾗﾝﾅｰ前ｽﾄｯﾊﾟｰ開条件2
6851  LD      M420  ; 連続起動
      AND     T230  ; ﾅｯﾄﾗﾝﾅｰ前ｽﾄｯﾊﾟｰ部ﾊﾟﾚｯﾄ検出
      AND     M291  ; ﾅｯﾄﾗﾝﾅｰ前ｽﾄｯﾊﾟｰ部ｽﾄｯﾊﾟｰ入端
      AND     M714  ; ﾅｯﾄﾗﾝﾅｰ前ｽﾄｯﾊﾟｰ開条件2
      OR      M715  ; ﾅｯﾄﾗﾝﾅｰ前ｽﾄｯﾊﾟｰ抜
      AND     M421  ; 連続運転
      ANI     M718  ; ﾅｯﾄﾗﾝﾅｰ前ｽﾄｯﾊﾟｰｻｲｸﾙ2完了
      ANI     M707  ; ﾅｯﾄﾗﾝﾅｰ前ｽﾄｯﾊﾟｰ部送り開始
      OUT     M715  ; ﾅｯﾄﾗﾝﾅｰ前ｽﾄｯﾊﾟｰ抜
6860  LDI     X245  ; ﾅｯﾄﾗﾝﾅｰ部ﾊﾟﾚｯﾄ検出
      AND     M292  ; ﾅｯﾄﾗﾝﾅｰ部ｽﾄｯﾊﾟｰ抜端
      OUT     T238 K2  ; ﾅｯﾄﾗﾝﾅｰ部ﾊﾟﾚｯﾄ無
6866  LD      T238  ; ﾅｯﾄﾗﾝﾅｰ部ﾊﾟﾚｯﾄ無
      OR      M716  ; ﾅｯﾄﾗﾝﾅｰ部ﾊﾟﾚｯﾄ通過中
      AND     M715  ; ﾅｯﾄﾗﾝﾅｰ前ｽﾄｯﾊﾟｰ抜
      OUT     M716  ; ﾅｯﾄﾗﾝﾅｰ部ﾊﾟﾚｯﾄ通過中
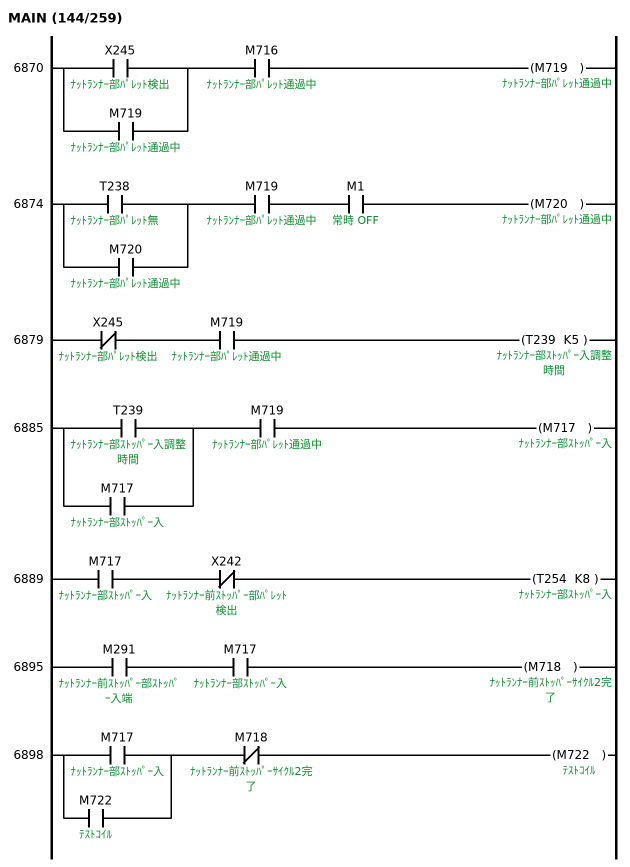
6870  LD      X245  ; ﾅｯﾄﾗﾝﾅｰ部ﾊﾟﾚｯﾄ検出
      OR      M719  ; ﾅｯﾄﾗﾝﾅｰ部ﾊﾟﾚｯﾄ通過中
      AND     M716  ; ﾅｯﾄﾗﾝﾅｰ部ﾊﾟﾚｯﾄ通過中
      OUT     M719  ; ﾅｯﾄﾗﾝﾅｰ部ﾊﾟﾚｯﾄ通過中
6874  LD      T238  ; ﾅｯﾄﾗﾝﾅｰ部ﾊﾟﾚｯﾄ無
      OR      M720  ; ﾅｯﾄﾗﾝﾅｰ部ﾊﾟﾚｯﾄ通過中
      AND     M719  ; ﾅｯﾄﾗﾝﾅｰ部ﾊﾟﾚｯﾄ通過中
      AND     M1  ; 常時 OFF
      OUT     M720  ; ﾅｯﾄﾗﾝﾅｰ部ﾊﾟﾚｯﾄ通過中
6879  LDI     X245  ; ﾅｯﾄﾗﾝﾅｰ部ﾊﾟﾚｯﾄ検出
      AND     M719  ; ﾅｯﾄﾗﾝﾅｰ部ﾊﾟﾚｯﾄ通過中
      OUT     T239 K5  ; ﾅｯﾄﾗﾝﾅｰ部ｽﾄｯﾊﾟｰ入調整時間
6885  LD      T239  ; ﾅｯﾄﾗﾝﾅｰ部ｽﾄｯﾊﾟｰ入調整時間
      OR      M717  ; ﾅｯﾄﾗﾝﾅｰ部ｽﾄｯﾊﾟｰ入
      AND     M719  ; ﾅｯﾄﾗﾝﾅｰ部ﾊﾟﾚｯﾄ通過中
      OUT     M717  ; ﾅｯﾄﾗﾝﾅｰ部ｽﾄｯﾊﾟｰ入
6889  LD      M717  ; ﾅｯﾄﾗﾝﾅｰ部ｽﾄｯﾊﾟｰ入
      ANI     X242  ; ﾅｯﾄﾗﾝﾅｰ前ｽﾄｯﾊﾟｰ部ﾊﾟﾚｯﾄ検出
      OUT     T254 K8  ; ﾅｯﾄﾗﾝﾅｰ部ｽﾄｯﾊﾟｰ入
6895  LD      M291  ; ﾅｯﾄﾗﾝﾅｰ前ｽﾄｯﾊﾟｰ部ｽﾄｯﾊﾟｰ入端
      AND     M717  ; ﾅｯﾄﾗﾝﾅｰ部ｽﾄｯﾊﾟｰ入
      OUT     M718  ; ﾅｯﾄﾗﾝﾅｰ前ｽﾄｯﾊﾟｰｻｲｸﾙ2完了
6898  LD      M717  ; ﾅｯﾄﾗﾝﾅｰ部ｽﾄｯﾊﾟｰ入
      OR      M722  ; ﾃｽﾄｺｲﾙ
      ANI     M718  ; ﾅｯﾄﾗﾝﾅｰ前ｽﾄｯﾊﾟｰｻｲｸﾙ2完了
      OUT     M722  ; ﾃｽﾄｺｲﾙ
